// RPC calls are not allowed in Local mode.
IF stat.bLocal THEN
	RPC_MoveAbs	:= M_SetRpcStatus(E_MOTOR_RPC_ERROR.LOCAL);
	RETURN;
// Move Absolute command is accepted only in OP state.
ELSIF	stat.nState <> E_MOTOR_STATE.OP	THEN
	RPC_MoveAbs	:= M_SetRpcStatus(E_MOTOR_RPC_ERROR.NOT_OP);
	RETURN;
// Set velocity cannot be <=0.0.
ELSIF	in_lrVel <= 0.0	THEN
	RPC_MoveAbs	:= M_SetRpcStatus(E_MOTOR_RPC_ERROR.VEL_NEG);
	RETURN;
// Set velocity cannot be greater than MAX Velocity.
ELSIF	in_lrVel > stat.axis.lrMaxVelocity	THEN
	RPC_MoveAbs	:= M_SetRpcStatus(E_MOTOR_RPC_ERROR.VEL_MAX);
	RETURN;
// If SW limits are active, check the limits
ELSIF cfg.lrMinPosition <> 0.0 OR cfg.lrMaxPosition <> 0.0 THEN
	IF in_lrPos < cfg.lrMinPosition THEN
		RPC_MoveAbs	:= M_SetRpcStatus(E_MOTOR_RPC_ERROR.SW_LIMIT_LOWER);
		RETURN;
	ELSIF in_lrPos > cfg.lrMaxPosition THEN
		RPC_MoveAbs	:= M_SetRpcStatus(E_MOTOR_RPC_ERROR.SW_LIMIT_UPPER);
		RETURN;
	END_IF
END_IF

// Set command
ctrl.nCommand 		:= E_MOTOR_COMMAND.MOTOR_MOVE;
ctrl.nMoveType		:= E_MOTOR_MOVE_TYPE.ABSOLUTE;
ctrl.lrPosition		:= in_lrPos;
ctrl.lrVelocity		:= in_lrVel;
ctrl.bExecute 		:= TRUE;

// Call was successful
RPC_MoveAbs	:= M_SetRpcStatus(E_MOTOR_RPC_ERROR.OK);
END_METHOD

{attribute 'TcRpcEnable':='1'}
METHOD RPC_MoveRel : INT
VAR_INPUT
	in_lrPos:	LREAL;
	in_lrVel:	LREAL;
END_VAR
// If unsafe, move is not allowed.
IF NOT in_bSafe THEN
	RPC_MoveRel	:= M_SetRpcStatus(E_MOTOR_RPC_ERROR.UNSAFE);
	RETURN;
END_IF

// RPC calls are not allowed in Local mode.
IF stat.bLocal THEN
	RPC_MoveRel	:= M_SetRpcStatus(E_MOTOR_RPC_ERROR.LOCAL);
	RETURN;
// Move Relative command is accepted only in OP state.
ELSIF	stat.nState <> E_MOTOR_STATE.OP	THEN
	RPC_MoveRel	:= M_SetRpcStatus(E_MOTOR_RPC_ERROR.NOT_OP);
	RETURN;
// Set velocity cannot be <=0.0.
ELSIF	in_lrVel <= 0.0	THEN
	RPC_MoveRel	:= M_SetRpcStatus(E_MOTOR_RPC_ERROR.VEL_NEG);
	RETURN;
// Set velocity cannot be greater than MAX Velocity.
ELSIF	in_lrVel > stat.axis.lrMaxVelocity	THEN
	RPC_MoveRel	:= M_SetRpcStatus(E_MOTOR_RPC_ERROR.VEL_MAX);
	RETURN;
// If SW limits are active, check the limits
ELSIF cfg.lrMinPosition <> 0.0 OR cfg.lrMaxPosition <> 0.0 THEN
	IF (in_lrPos + stat.lrPosActual) < cfg.lrMinPosition THEN
		RPC_MoveRel	:= M_SetRpcStatus(E_MOTOR_RPC_ERROR.SW_LIMIT_LOWER);
		RETURN;
	ELSIF (in_lrPos + stat.lrPosActual) > cfg.lrMaxPosition THEN
		RPC_MoveRel	:= M_SetRpcStatus(E_MOTOR_RPC_ERROR.SW_LIMIT_UPPER);
		RETURN;
	END_IF
END_IF

// Set command
ctrl.nCommand 		:= E_MOTOR_COMMAND.MOTOR_MOVE;
ctrl.nMoveType		:= E_MOTOR_MOVE_TYPE.RELATIVE;
ctrl.lrOffset		:= in_lrPos;
ctrl.lrVelocity		:= in_lrVel;
ctrl.bExecute 		:= TRUE;

// Call was successful
RPC_MoveRel	:= M_SetRpcStatus(E_MOTOR_RPC_ERROR.OK);
END_METHOD

{attribute 'TcRpcEnable':='1'}
METHOD RPC_MoveVel : INT
VAR_INPUT
	in_lrVel:	LREAL;
END_VAR
// If unsafe, move is not allowed.
IF NOT in_bSafe THEN
	RPC_MoveVel	:= M_SetRpcStatus(E_MOTOR_RPC_ERROR.UNSAFE);
	RETURN;
END_IF

// RPC calls are not allowed in Local mode.
IF stat.bLocal THEN
	RPC_MoveVel	:= M_SetRpcStatus(E_MOTOR_RPC_ERROR.LOCAL);
	RETURN;
END_IF

// Move in Velocity command is accepted only in OP state.
IF	stat.nState <> E_MOTOR_STATE.OP	THEN
	RPC_MoveVel	:= M_SetRpcStatus(E_MOTOR_RPC_ERROR.NOT_OP);
	RETURN;
// Set velocity cannot be 0.0.
ELSIF	in_lrVel = 0.0	THEN
	RPC_MoveVel	:= M_SetRpcStatus(E_MOTOR_RPC_ERROR.VEL_ZERO);
	RETURN;
// Set velocity cannot be greater than MAX Velocity.
// Note that MoveVel() accepts negative velocity. That is
// why we use ABS().
ELSIF	ABS(in_lrVel) > stat.axis.lrMaxVelocity	THEN
	RPC_MoveVel	:= M_SetRpcStatus(E_MOTOR_RPC_ERROR.VEL_MAX);
	RETURN;
ELSE
	// Set command
	ctrl.nCommand 		:= E_MOTOR_COMMAND.MOTOR_MOVE;
	ctrl.nMoveType		:= E_MOTOR_MOVE_TYPE.VELOCITY;
	
	// Set the direction of movement based on the velocity sign.
	// Velocity is always passed as positive.
	IF in_lrVel < 0.0 THEN
		ctrl.lrVelocity		:= -in_lrVel;
		ctrl.nDirection		:= MC_Negative_Direction;
	ELSE
		ctrl.lrVelocity		:= in_lrVel;
		ctrl.nDirection		:= MC_Positive_Direction;
	END_IF

	ctrl.bExecute 		:= TRUE;
	
	// Call was successful
	RPC_MoveVel	:= M_SetRpcStatus(E_MOTOR_RPC_ERROR.OK);
END_IF
END_METHOD

{attribute 'TcRpcEnable':='1'}
METHOD RPC_Reset : INT
VAR_INPUT
END_VAR
// RPC calls are not allowed in Local mode.
IF stat.bLocal THEN
	RPC_Reset	:= M_SetRpcStatus(E_MOTOR_RPC_ERROR.LOCAL);
	RETURN;
END_IF

ctrl.nCommand := E_MOTOR_COMMAND.RESET;
ctrl.bExecute := TRUE;

// Call was successful
RPC_Reset	:= M_SetRpcStatus(E_MOTOR_RPC_ERROR.OK);
END_METHOD

{attribute 'TcRpcEnable':='1'}
METHOD RPC_SetDebug : INT
VAR_INPUT
	in_bDebug:	BOOL 	:= FALSE;		// If TRUE, show event logs of Debug type
END_VAR
// Enable/disable Debugging
cfg.bDebug	:= in_bDebug;

// Call was successful
RPC_SetDebug	:= M_SetRpcStatus(E_MOTOR_RPC_ERROR.OK);
END_METHOD

{attribute 'TcRpcEnable':='1'}
METHOD RPC_SetLog : INT
VAR_INPUT
	in_bLog:	BOOL 	:= FALSE;		// If TRUE, activate event logging
END_VAR
// Enable/disable Logging
cfg.bLog	:= in_bLog;

// Call was successful
RPC_SetLog	:= M_SetRpcStatus(E_MOTOR_RPC_ERROR.OK);
END_METHOD

{attribute 'TcRpcEnable':='1'}
METHOD RPC_Stop : INT
VAR_INPUT
END_VAR
// RPC calls are not allowed in Local mode.
IF stat.bLocal THEN
	RPC_Stop	:= M_SetRpcStatus(E_MOTOR_RPC_ERROR.LOCAL);
	RETURN;
END_IF

ctrl.nCommand := E_MOTOR_COMMAND.STOP;
ctrl.bExecute := TRUE;

// Call was successful
RPC_Stop	:= M_SetRpcStatus(E_MOTOR_RPC_ERROR.OK);
END_METHOD

METHOD UserPostInit : BOOL
VAR_OUTPUT
	nErrorId:	E_MOTOR_ERROR	:= E_MOTOR_ERROR.OK;
END_VAR
VAR
END_VAR
// TODOUSER:
// Dummy implementation.
// Configure cfg.bExecUserPostInit to TRUE.
// Implement PostInit logic.
// If error, set error description in this method using M_SetError(nErrorId, ...) - see below.

stat.sStatus	:= 'User Post-Init Method';

IF Dummy_UserExample() THEN
	UserPostInit	:= TRUE;
	stat.sStatus	:= 'OK';
	RETURN;
END_IF

// Check if the timer has expired. If yes, we have a problem *)
toutCmd();
IF toutCmd.Q = TRUE THEN
	toutCmd(IN := FALSE);
	nErrorId := E_MOTOR_ERROR.TIMEOUT_USER_POSTINIT;
	M_SetError(nErrorId, 'ERROR: Timeout during USER POST INIT');
	UserPostInit	:= TRUE;	// Exit (with error)
	RETURN;
END_IF


(* Check for motion errors *)
IF Axis.Status.Error THEN
	nErrorId	:= UDINT_TO_INT(Axis.Status.ErrorID);
	M_SetError(nErrorId, 'ERROR: Axis error during USER POST INIT');
	UserPostInit	:= TRUE;	// Exit (with error)
	RETURN;
END_IF

// Dummy implementation.
// Dummy error for testing.
//nErrorId := E_MOTOR_ERROR.TIMEOUT;
//M_SetError(nErrorId, 'ERROR: Dummy error during USER POST INIT');
//UserPostInit	:= TRUE;
RETURN;
END_METHOD

METHOD UserPostMove : BOOL
VAR_OUTPUT
	nErrorId:	E_MOTOR_ERROR	:= E_MOTOR_ERROR.OK;
END_VAR
VAR
END_VAR
// TODOUSER:
// Dummy implementation.
// Configure cfg.bExecUserPostMove to TRUE.
// Implement PostMove logic.
// If error, set error description in this method using M_SetError(nErrorId, ...) - see below.

stat.sStatus	:= 'User Post-Move Method';

IF Dummy_UserExample() THEN
	UserPostMove	:= TRUE;
	stat.sStatus	:= 'OK';
	RETURN;
END_IF

// Check if the timer has expired. If yes, we have a problem *)
toutCmd();
IF toutCmd.Q = TRUE THEN
	toutCmd(IN := FALSE);
	nErrorId := E_MOTOR_ERROR.TIMEOUT_USER_POSTMOVE;
	M_SetError(nErrorId, 'ERROR: Timeout during USER POST MOVE');
	UserPostMove	:= TRUE;	// Exit (with error)
	RETURN;
END_IF


(* Check for motion errors *)
IF Axis.Status.Error THEN
	nErrorId	:= UDINT_TO_INT(Axis.Status.ErrorID);
	M_SetError(nErrorId, 'ERROR: Axis error during USER POST MOVE');
	UserPostMove	:= TRUE;	// Exit (with error)
	RETURN;
END_IF

// Dummy implementation.
// Dummy error for testing.
//nErrorId := E_MOTOR_ERROR.TIMEOUT;
//M_SetError(nErrorId, 'ERROR: Dummy error during USER POST MOVE');
//UserPostMove	:= TRUE;
RETURN;
END_METHOD

METHOD UserPreInit : BOOL
VAR_OUTPUT
	nErrorId:	E_MOTOR_ERROR	:= E_MOTOR_ERROR.OK;
END_VAR
VAR
END_VAR
// TODOUSER:
// Dummy implementation.
// Configure cfg.bExecUserPreInit to TRUE.
// Implement PreInit logic.
// If error, set error description in this method using M_SetError(nErrorId, ...) - see below.

stat.sStatus	:= 'User Pre-Init Method';

IF Dummy_UserExample() THEN
	UserPreInit	:= TRUE;
	stat.sStatus	:= 'OK';
	RETURN;
END_IF

// Check if the timer has expired. If yes, we have a problem *)
toutCmd();
IF toutCmd.Q = TRUE THEN
	toutCmd(IN := FALSE);
	nErrorId := E_MOTOR_ERROR.TIMEOUT_USER_PREINIT;
	M_SetError(nErrorId, 'ERROR: Timeout during USER PRE INIT');
	UserPreInit	:= TRUE;	// Exit (with error)
	RETURN;
END_IF


(* Check for motion errors *)
IF Axis.Status.Error THEN
	nErrorId	:= UDINT_TO_INT(Axis.Status.ErrorID);
	M_SetError(nErrorId, 'ERROR: Axis error during USER PRE INIT');
	UserPreInit	:= TRUE;	// Exit (with error)
	RETURN;
END_IF

// Dummy implementation.
// Dummy error for testing.
//nErrorId := E_MOTOR_ERROR.TIMEOUT;
//M_SetError(nErrorId, 'ERROR: Dummy error during USER PRE INIT');
//UserPreInit	:= TRUE;
RETURN;
END_METHOD

METHOD UserPreMove : BOOL
VAR_OUTPUT
	nErrorId:	E_MOTOR_ERROR	:= E_MOTOR_ERROR.OK;
END_VAR
VAR
END_VAR
// TODOUSER:
// Dummy implementation.
// Configure cfg.bExecUserPreMove to TRUE.
// Implement PreMove logic.
// If error, set error description in this method using M_SetError(nErrorId, ...) - see below.

stat.sStatus	:= 'User Pre-Move Method';

IF Dummy_UserExample() THEN
	UserPreMove		:= TRUE;
	stat.sStatus	:= 'OK';
	RETURN;
END_IF

// Check if the timer has expired. If yes, we have a problem *)
toutCmd();
IF toutCmd.Q = TRUE THEN
	toutCmd(IN := FALSE);
	nErrorId := E_MOTOR_ERROR.TIMEOUT_USER_PREMOVE;
	M_SetError(nErrorId, 'ERROR: Timeout during USER PRE MOVE');
	UserPreMove	:= TRUE;	// Exit (with error)
	RETURN;
END_IF


(* Check for motion errors *)
IF Axis.Status.Error THEN
	nErrorId	:= UDINT_TO_INT(Axis.Status.ErrorID);
	M_SetError(nErrorId, 'ERROR: Axis error during USER PRE MOVE');
	UserPreMove	:= TRUE;	// Exit (with error)
	RETURN;
END_IF

// Dummy implementation.
// Dummy error for testing.
//nErrorId := E_MOTOR_ERROR.TIMEOUT;
//M_SetError(nErrorId, 'ERROR: Dummy error during USER PRE MOVE');
//UserPreMove	:= TRUE;
RETURN;
END_METHOD

END_FUNCTION_BLOCK

// ---- POUs/Motor/FB_MOTOR_BASE.TcPOU
FUNCTION_BLOCK FB_MOTOR_BASE
VAR_INPUT
	// EICSSW-1923
	{attribute 'OPC.UA.DA' := '0'}
	in_bSafe:		BOOL	:= TRUE;	// Flag if safe to move the motor
	{attribute 'OPC.UA.DA' := '0'}
	in_bDisableIfUnsafe:	BOOL := FALSE;	// If unsafe, motor is disabled
END_VAR
VAR_OUTPUT
END_VAR
VAR RETAIN
END_VAR
VAR
	{attribute 'OPC.UA.DA' := '1'}
	cfg:		T_MOTOR_CFG;		// Config parameters
	{attribute 'OPC.UA.DA' := '1'}
	ctrl:		T_MOTOR_CTRL;		// Control parameters
	{attribute 'OPC.UA.DA' := '1'}
	{attribute 'OPC.UA.DA.Access' := '1'}
	info:		T_MOTOR_INFO;		// Driver Info - ReadOnly
	{attribute 'OPC.UA.DA' := '1'}
	{attribute 'OPC.UA.DA.Access' := '1'}
	stat:		T_MOTOR_STAT;		// Status parameters - ReadOnly

	{attribute 'OPC.UA.DA' := '0'}
	nEvent:		      	DINT := E_MOTOR_EVENT.NONE;
	{attribute 'OPC.UA.DA' := '0'}
	nInternalEvent:		DINT := E_MOTOR_EVENT.NONE;
	
	// Operational Events
	{attribute 'OPC.UA.DA' := '0'}
	fbEventStart:	FB_TcMessage;
	{attribute 'OPC.UA.DA' := '0'}
	fbEventEnd:		FB_TcMessage;
	{attribute 'OPC.UA.DA' := '0'}
	fbEventError:	FB_TcMessage;
	{attribute 'OPC.UA.DA' := '0'}
	fbEventDebug:	FB_TcMessage;
	{attribute 'OPC.UA.DA' := '0'}
	fbEventGeneral:	FB_TcMessage;
	{attribute 'OPC.UA.DA' := '0'}
	fbEventMoveAbs:	FB_TcMessage;
	{attribute 'OPC.UA.DA' := '0'}
	fbEventMoveRel:	FB_TcMessage;
	{attribute 'OPC.UA.DA' := '0'}
	fbEventMoveVel:	FB_TcMessage;
	
	(***** Physical signals - to be mapped!!! *****)

	(* Outputs *)

	(* Inputs *)
	

END_VAR

METHOD ActionClearNOVRAM
VAR_INPUT
END_VAR
END_METHOD

METHOD ActionEnableExecute
VAR_INPUT
END_VAR
END_METHOD

METHOD ActionErrExecute
VAR
END_VAR
END_METHOD

METHOD ActionInitAbort
VAR_INPUT
END_VAR
END_METHOD

METHOD ActionInitComplete
VAR_INPUT
END_VAR
END_METHOD

METHOD ActionInitExecute
VAR_INPUT
END_VAR
END_METHOD

METHOD ActionInitReject
VAR_INPUT
END_VAR
END_METHOD

METHOD ActionMoveExecute
VAR_INPUT
END_VAR
END_METHOD

METHOD ActionResetExecute
VAR_INPUT
END_VAR
END_METHOD

METHOD ActionSetPosition
VAR_INPUT
END_VAR
END_METHOD

METHOD ActionStopExecute
VAR_INPUT
END_VAR
END_METHOD

METHOD ActionUnexpExecute
VAR_INPUT
END_VAR
END_METHOD

METHOD ActivityClearingNOVRAM
VAR_INPUT
END_VAR
END_METHOD

METHOD ActivityInitAborting
VAR_INPUT
END_VAR
END_METHOD

METHOD ActivityInitializing
VAR_INPUT
END_VAR
END_METHOD

METHOD ActivityMoving
VAR_INPUT
END_VAR
END_METHOD

METHOD ActivitySettingPosition
VAR_INPUT
END_VAR
END_METHOD

METHOD ActivityStopping
VAR_INPUT
END_VAR
END_METHOD

METHOD CheckForEvents
VAR_INPUT
END_VAR
END_METHOD

METHOD M_CheckDisableIfUnsafe
VAR_INPUT
END_VAR
IF NOT in_bSafe AND in_bDisableIfUnsafe	THEN
	IF stat.bEnabled	THEN
		stat.bEnabled	:= FALSE;
		M_LogEventGeneral('Not safe to move. Motor disabled.');
	END_IF
END_IF
END_METHOD

METHOD M_GetErrorText : STRING
VAR_INPUT
	nErrorID:	DINT;
END_VAR
VAR
	str:	STRING;
END_VAR
			
CASE nErrorID OF
	E_MOTOR_ERROR.OK:						str	:= 'OK';
	E_MOTOR_ERROR.HW_NOT_OP:				str	:= 'ERROR: TwinCAT not OP or CouplerState not mapped.';
	E_MOTOR_ERROR.LOCAL:					str	:= 'ERROR: Control not allowed. Motor in Local mode.';
	E_MOTOR_ERROR.INIT_ABORTED:				str	:= 'ERROR: INIT command aborted.';
	E_MOTOR_ERROR.TIMEOUT_INIT:				str	:= 'ERROR: INIT timed out.';
	E_MOTOR_ERROR.TIMEOUT_MOVE:				str	:= 'ERROR: Move timed out.';
	E_MOTOR_ERROR.TIMEOUT_RESET:			str	:= 'ERROR: Reset timed out.';
	E_MOTOR_ERROR.TIMEOUT_SETPOS:			str	:= 'ERROR: Set Position timed out.';
	E_MOTOR_ERROR.TIMEOUT_USER_PREINIT:		str	:= 'ERROR: User PRE-INIT timed out.';
	E_MOTOR_ERROR.TIMEOUT_USER_POSTINIT:	str	:= 'ERROR: User POST-INIT timed out.';
	E_MOTOR_ERROR.TIMEOUT_USER_PREMOVE:		str	:= 'ERROR: User PRE-MOVE timed out.';
	E_MOTOR_ERROR.TIMEOUT_USER_POSTMOVE:	str	:= 'ERROR: User POST-MOVE timed out.';
	E_MOTOR_ERROR.SETPOS:					str	:= 'ERROR: Set Position failed.';
	E_MOTOR_ERROR.STOP:						str	:= 'ERROR: STOP failed.';
	
	E_MOTOR_ERROR.ABORT:					str	:= 'ERROR: Motion aborted.';
	E_MOTOR_ERROR.SW_LIMIT_LOWER:			str	:= 'ERROR: Lower SW Limit Exceeded.';
	E_MOTOR_ERROR.SW_LIMIT_UPPER:			str	:= 'ERROR: Upper SW Limit Exceeded.';
	E_MOTOR_ERROR.BRAKE_ACTIVE:				str	:= 'ERROR: Cannot move. Brake active.';
	E_MOTOR_ERROR.BRAKE_ENGAGE:				str	:= 'ERROR: Failed to engage brake.';
	E_MOTOR_ERROR.BRAKE_DISENGAGE:			str	:= 'ERROR: Failed to disengage brake.';
	E_MOTOR_ERROR.SWITCH_NOT_USED:			str	:= 'ERROR: Switch was not detected in previous INIT action.';
	E_MOTOR_ERROR.ENABLE:					str	:= 'ERROR: Failed to enable Axis.';
	E_MOTOR_ERROR.NOVRAM_READ:				str	:= 'ERROR: Failed to read from NOVRAM';
	E_MOTOR_ERROR.NOVRAM_WRITE:				str	:= 'ERROR: Failed to write to NOVRAM';
	E_MOTOR_ERROR.SWITCH_EXIT:				str	:= 'ERROR: Timeout on switch exit. Check nTimeoutSwitch.';
	E_MOTOR_ERROR.STOP_LIMITS_BOTH:			str	:= 'ERROR: Both LSTOP and USTOP limits active.';
	E_MOTOR_ERROR.HW_LIMITS_BOTH:			str	:= 'ERROR: Both limit switches LHW and UHW active.';
	E_MOTOR_ERROR.IN_POS:					str	:= 'ERROR: In-Pos switch not active at the end of movement.';
	E_MOTOR_ERROR.LOCKED:					str	:= 'ERROR: Motor Locked! Cannot move.';
	E_MOTOR_ERROR.SoE_ADS_ERROR:			str	:= 'ERROR: SoE ADS Error.';
	E_MOTOR_ERROR.SoE_SERCOS_ERROR:			str	:= 'ERROR: SoE Sercos Error.';
	E_MOTOR_ERROR.UNSAFE:					str	:= 'ERROR: Not safe to move.';

	E_MOTOR_ERROR.SIM_NOT_INITIALISED:		str	:= 'ERROR: Simulator not initialised.';
	E_MOTOR_ERROR.SIM_NULL_POINTER:			str	:= 'ERROR: Simulator input parameter is a NULL pointer.';
	
	// Beckhoff TwinCAT most common errors
	E_MOTOR_ERROR.TC_VEL:					str	:= 'ERROR: Requested set velocity is not allowed.';
	E_MOTOR_ERROR.TC_NOT_READY_FOR_START:	str	:= 'ERROR: Drive not ready during axis start.';
	E_MOTOR_ERROR.TC_DISABLED_MOVE:			str	:= 'ERROR: Motor disabled while moving. Reset required!';
	E_MOTOR_ERROR.TC_BISECTION:				str	:= 'WARNING: Motion command could not be realized (BISECTION)';
	E_MOTOR_ERROR.TC_MODULO_POS:			str	:= 'ERROR: Target position >= full turn (modulo-period)';
	E_MOTOR_ERROR.TC_STOP_ACTIVE:			str	:= 'ERROR: Stop command still active. Axis locked. Reset required!';
	E_MOTOR_ERROR.TC_VEL_NEG:				str	:= 'ERROR: Set velocity not allowed (<=0)';
	E_MOTOR_ERROR.TC_TARGET_LSW:			str	:= 'ERROR: Target position beyond Lower Software Limit.';
	E_MOTOR_ERROR.TC_TARGET_USW:			str	:= 'ERROR: Target position beyond Upper Software Limit.';
	E_MOTOR_ERROR.TC_FOLLOWING_ERROR:		str	:= 'ERROR: Following error. Reset required!';
	E_MOTOR_ERROR.TC_NOT_READY:				str	:= 'ERROR: Drive not ready for operation.';
	E_MOTOR_ERROR.TC_IN_POS_6_SEC:			str	:= 'ERROR: In-position 6 sec timeout. Reset required!';
ELSE
	IF nErrorID > 10000 THEN
		str	:= concat('Unregistered error: ', DINT_TO_STRING(nErrorID));
		str	:= concat(str, ' Check TwinCAT error codes.');
	ELSE
		str	:= 'Unregistered internal error. Report it to ESO.';
	END_IF
END_CASE

M_GetErrorText	:= str;
END_METHOD

METHOD M_GetLogicalState : BOOL
(*
	This method returns the state of the variable based on its 
	activeLow configuration.
	Syntax:
		bState	:= GetLogicalState (<var value>,  <activeLow cfg>);
		
	Example 1:
		var = TRUE;
		activeLow = FALSE;
		bState	:= GetLogicalState (TRUE,  FALSE); = TRUE

	Example 2:
		var = TRUE;
		activeLow = TRUE;
		bState	:= GetLogicalState (TRUE,  TRUE); = FALSE
*)
VAR_INPUT
	state:		BOOL;
	activeLow:	BOOL;
END_VAR
IF activeLow THEN
	M_GetLogicalState := NOT state;
ELSE
	M_GetLogicalState := state;
END_IF
END_METHOD

METHOD M_GetTimeInSec : UDINT
(*
	This method returns absolute time in seconds.
*)
VAR_INPUT
END_VAR
VAR
	fbGetSystemTime:	GETSYSTEMTIME;
	timeLoDW:			DWORD;
	timeHiDW:			DWORD;
	nSecondsLo:			UDINT;
	nSecondsHi:			UDINT;

END_VAR
fbGetSystemTime (timeLoDW => timeLoDW, timeHiDW => timeHiDW); (* System time is given in 100ns *)
nSecondsLo	:= DWORD_TO_UDINT(timeLoDW) / 10000000; (* Convert to seconds *)
(* One unit from HI WORD represents 16#FFFFFFFF/10000000 = 429.4967296 seconds *)
nSecondsHi	:= LREAL_TO_UDINT(DWORD_TO_LREAL(timeHiDW) * 429.4967296);

M_GetTimeInSec	:= nSecondsHi + nSecondsLo;
END_METHOD

METHOD M_LogEventDebug : BOOL
VAR_INPUT
	sText:	STRING	:= '';
END_VAR
// Log Debug events only if both logging and debugging are enabled AND it is not a tracking command
IF cfg.bLog AND cfg.bDebug AND NOT (ctrl.nMoveType = E_MOTOR_MOVE_TYPE.TRACKING) THEN
	fbEventDebug.ipArguments.Clear().AddString(sText);
	fbEventDebug.Send(0);
END_IF
END_METHOD

METHOD M_LogEventEnd : BOOL
VAR_INPUT
	sText:	STRING	:= '';
END_VAR
// Log only if logging is enabled AND it is not a tracking command
IF  NOT cfg.bLog OR ctrl.nMoveType = E_MOTOR_MOVE_TYPE.TRACKING THEN
	RETURN;
END_IF

fbEventEnd.ipArguments.Clear().AddString(sText);
fbEventEnd.Send(0);
END_METHOD

METHOD M_LogEventError : BOOL
VAR_INPUT
	sText:	STRING	:= '';
END_VAR
// Log only if logging is enabled
IF  NOT cfg.bLog THEN
	RETURN;
END_IF

fbEventError.ipArguments.Clear().AddString(sText);
fbEventError.Send(0);
END_METHOD

METHOD M_LogEventGeneral : BOOL
VAR_INPUT
	sText:	STRING	:= '';
END_VAR
// Log only if logging is enabled AND it is not a tracking command
IF  NOT cfg.bLog OR ctrl.nMoveType = E_MOTOR_MOVE_TYPE.TRACKING THEN
	RETURN;
END_IF

fbEventGeneral.ipArguments.Clear().AddString(sText);
fbEventGeneral.Send(0);
END_METHOD

METHOD M_LogEventMoveAbs : BOOL
VAR_INPUT
	lrPos:	LREAL;
	lrVel:	LREAL;
END_VAR
// Log only if logging is enabled AND it is not a tracking command
IF  NOT cfg.bLog OR ctrl.nMoveType = E_MOTOR_MOVE_TYPE.TRACKING THEN
	RETURN;
END_IF

fbEventMoveAbs.ipArguments.Clear().AddLReal(lrPos).AddLReal(lrVel);
fbEventMoveAbs.Send(0);
END_METHOD

METHOD M_LogEventMoveRel : BOOL
VAR_INPUT
	lrPosRel:	LREAL;
	lrPosAct:	LREAL;
	lrVel:		LREAL;
END_VAR
// Log only if logging is enabled AND it is not a tracking command
IF  NOT cfg.bLog OR ctrl.nMoveType = E_MOTOR_MOVE_TYPE.TRACKING THEN
	RETURN;
END_IF

fbEventMoveRel.ipArguments.Clear().AddLReal(lrPosRel).AddLReal(lrPosAct).AddLReal(lrVel);
fbEventMoveRel.Send(0);
END_METHOD

METHOD M_LogEventMoveVel : BOOL
VAR_INPUT
	lrVel:	LREAL;
	dir:	DINT;
END_VAR
VAR
	lrVelTmp:	LREAL;
END_VAR
// Log only if logging is enabled AND it is not a tracking command
IF  NOT cfg.bLog OR ctrl.nMoveType = E_MOTOR_MOVE_TYPE.TRACKING THEN
	RETURN;
END_IF

IF dir = MC_Negative_Direction THEN
	lrVelTmp	:= -lrVel;
ELSE
	lrVelTmp	:= +lrVel;
END_IF
fbEventMoveVel.ipArguments.Clear().AddLReal(lrVelTmp);
fbEventMoveVel.Send(0);
END_METHOD

METHOD M_LogEventStart : BOOL
VAR_INPUT
	sText:	STRING	:= '';
END_VAR
// Log only if logging is enabled AND it is not a tracking command
IF  NOT cfg.bLog OR ctrl.nMoveType = E_MOTOR_MOVE_TYPE.TRACKING THEN
	RETURN;
END_IF

fbEventStart.ipArguments.Clear().AddString(sText);
fbEventStart.Send(0);
END_METHOD

// This method copies the description of the first error that caused the failure.
// For example, in case of a failure during move, the error description
// is written into stat.sFirstError and then the motor is commanded to stop.
// At the end of the stop, stat.sFirstError will be copied into stat.sErrorText so
// the user can see the real reason for the failure.
METHOD M_ReportFirstError
VAR_INPUT
END_VAR
IF stat.sFirstError <> '' THEN
	stat.sErrorText	:= stat.sFirstError;	// Copy stored error
	stat.sFirstError:= '';					// Clear stored error
END_IF
END_METHOD

METHOD M_SetStatus
VAR_INPUT
	nErrorCode:	E_MOTOR_ERROR;
END_VAR
stat.nErrorCode 	:= nErrorCode;
stat.sErrorText 	:= M_GetErrorText(nErrorCode);

IF nErrorCode <> E_MOTOR_ERROR.OK THEN
	stat.sStatus	:= 'ERROR';
	stat.nStatus	:= E_MOTOR_STATUS.ERROR;
ELSE
	stat.sStatus	:= 'OK';
	stat.nStatus	:= E_MOTOR_STATUS.OK;
END_IF
END_METHOD

METHOD M_SetStatusDescription
VAR_INPUT
	nAxisStatus:	E_MOTOR_STATUS;	(* Status number *)
	sStatus:		STRING;			(* Status text, e.g. IDLE, BUSY, etc. *)
END_VAR
stat.nErrorCode		:= E_MOTOR_ERROR.OK;
stat.nStatus		:= nAxisStatus;
stat.sErrorText		:= 'OK';
stat.sStatus		:= sStatus;
END_METHOD

METHOD ProcessEvents
VAR_INPUT
END_VAR

VAR
END_VAR

(* 
	Before processing the event, execute the Do-Activity tasks. 
	Note that, in case of orthogonal regions, more than one Do-Activity 
	could run in the same PLC cycle.
	Note: Most of these activities have timeouts since they take time.
*)

IF stat.nSubstate = E_MOTOR_SUBSTATE.NOTOP_INITIALIZING THEN
	ActivityInitializing();
END_IF

IF stat.nSubstate = E_MOTOR_SUBSTATE.NOTOP_ABORTING THEN
	ActivityInitAborting();
END_IF

IF stat.nSubstate = E_MOTOR_SUBSTATE.NOTOP_CLEARING_NOVRAM THEN
	ActivityClearingNOVRAM();
END_IF

IF	stat.nSubstate = E_MOTOR_SUBSTATE.OP_MOVING	AND
	nEvent <> E_MOTOR_EVENT.STOP					THEN
	ActivityMoving();
END_IF

IF stat.nSubstate = E_MOTOR_SUBSTATE.OP_STOPPING THEN
	ActivityStopping();
END_IF

IF stat.nSubstate = E_MOTOR_SUBSTATE.OP_SETTING_POS THEN
	ActivitySettingPosition();
END_IF


(* 
	Evaluate state machine transitions.
*)

CASE stat.nState OF

//***********************************
// NOTOP
//***********************************
E_MOTOR_STATE.NOTOP:

	(* Transitions from NOTOP substates *)
	CASE stat.nSubstate OF
	
	E_MOTOR_SUBSTATE.NOTOP_NOTREADY:		
		// Update error description if pending.
		M_ReportFirstError();		
		IF nEvent = E_MOTOR_EVENT.RESET THEN
			ActionResetExecute();
			RETURN;
		ELSIF nEvent = E_MOTOR_EVENT.INIT THEN
			ActionInitExecute();
			M_SetStatus(E_MOTOR_ERROR.OK);
			SetState(E_MOTOR_STATE.NOTOP, E_MOTOR_SUBSTATE.NOTOP_INITIALIZING);
			RETURN;
		ELSIF nEvent = E_MOTOR_EVENT.CLEAR_NOVRAM THEN
			ActionClearNOVRAM();
			M_SetStatus(E_MOTOR_ERROR.OK);
			SetState(E_MOTOR_STATE.NOTOP, E_MOTOR_SUBSTATE.NOTOP_CLEARING_NOVRAM);
			RETURN;
		END_IF
		
	E_MOTOR_SUBSTATE.NOTOP_INITIALIZING:			
		IF nEvent = E_MOTOR_EVENT.UNSAFE THEN
			// Set the first error that caused the failure
			M_SetStatus(E_MOTOR_ERROR.UNSAFE);
			stat.sFirstError	:= M_GetErrorText(E_MOTOR_ERROR.UNSAFE);
			M_LogEventError(stat.sFirstError);
			ActionInitAbort();
			SetState(E_MOTOR_STATE.NOTOP, E_MOTOR_SUBSTATE.NOTOP_ABORTING);
			RETURN;
		END_IF

		IF 	nEvent = E_MOTOR_EVENT.STOP  	OR  
			nEvent = E_MOTOR_EVENT.RESET 	 	THEN
			ActionInitAbort();
			SetState(E_MOTOR_STATE.NOTOP, E_MOTOR_SUBSTATE.NOTOP_ABORTING);
			RETURN;
		ELSIF nEvent = E_MOTOR_EVENT.ERRINIT THEN
			// Error description is set in ActivityInitializing().
			SetState(E_MOTOR_STATE.NOTOP, E_MOTOR_SUBSTATE.NOTOP_ERROR);
			RETURN;
		ELSIF nEvent = E_MOTOR_EVENT.ERRBRAKE OR 
			  nEvent = E_MOTOR_EVENT.ERRRESET 	THEN
			SetState(E_MOTOR_STATE.NOTOP, E_MOTOR_SUBSTATE.NOTOP_ERROR);
			RETURN;
		ELSIF nEvent = E_MOTOR_EVENT.INITDONE THEN
			ActionInitComplete();
			SetState(E_MOTOR_STATE.NOTOP, E_MOTOR_SUBSTATE.NOTOP_READY);
			RETURN;
		END_IF
		
	E_MOTOR_SUBSTATE.NOTOP_ABORTING:			
		IF	nEvent = E_MOTOR_EVENT.STOPDONE OR 
			nEvent = E_MOTOR_EVENT.ERRSTOP 		THEN
			SetState(E_MOTOR_STATE.NOTOP, E_MOTOR_SUBSTATE.NOTOP_NOTREADY);
			RETURN;
		ELSIF nEvent = E_MOTOR_EVENT.RESET THEN
			ActionInitAbort();
			M_SetStatus(E_MOTOR_ERROR.OK);
			SetState(E_MOTOR_STATE.NOTOP, E_MOTOR_SUBSTATE.NOTOP_NOTREADY);
			RETURN;
		END_IF
		
	E_MOTOR_SUBSTATE.NOTOP_READY:			
		// Check if the motor should be disabled due to non-safe operation
		M_CheckDisableIfUnsafe();
	
		IF nEvent = E_MOTOR_EVENT.RESET THEN
			ActionResetExecute();
			SetState(E_MOTOR_STATE.NOTOP, E_MOTOR_SUBSTATE.NOTOP_NOTREADY);
			RETURN;
		ELSIF nEvent = E_MOTOR_EVENT.ERRFAULT THEN
			SetState(E_MOTOR_STATE.NOTOP, E_MOTOR_SUBSTATE.NOTOP_NOTREADY);			
			RETURN;
		ELSIF nEvent = E_MOTOR_EVENT.ENABLE THEN
			M_LogEventGeneral('ENABLE Executed');
			M_SetStatus(E_MOTOR_ERROR.OK);
			SetState(E_MOTOR_STATE.OP, E_MOTOR_SUBSTATE.OP_STANDSTILL);
			RETURN;
		END_IF

	E_MOTOR_SUBSTATE.NOTOP_ERROR:			
		// Update error description if pending.
		M_ReportFirstError();		
		// Check if the motor should be disabled due to non-safe operation
		M_CheckDisableIfUnsafe();
	
		IF nEvent = E_MOTOR_EVENT.RESET THEN
			ActionResetExecute();
			SetState(E_MOTOR_STATE.NOTOP, E_MOTOR_SUBSTATE.NOTOP_NOTREADY);
			RETURN;
		ELSIF nEvent = E_MOTOR_EVENT.INIT THEN
			ActionInitExecute();
			M_SetStatus(E_MOTOR_ERROR.OK);
			SetState(E_MOTOR_STATE.NOTOP, E_MOTOR_SUBSTATE.NOTOP_INITIALIZING);
			RETURN;
		END_IF
		
	END_CASE

	(* Transitions from NOTOP state *)
	IF nEvent = E_MOTOR_EVENT.STOP THEN
		// Nothing to do. Motor is already standing
		RETURN;
	ELSIF nEvent = E_MOTOR_EVENT.ERRHW THEN
		stat.bEnabled		:= FALSE;	// Disable motor
		stat.bInitialised	:= FALSE;	// The motor has to be re-initialised
		SetState(E_MOTOR_STATE.NOTOP, E_MOTOR_SUBSTATE.NOTOP_ERROR);
		RETURN;
	ELSIF nEvent = E_MOTOR_EVENT.ERRLOCAL THEN
		M_SetStatus(E_MOTOR_ERROR.LOCAL);
		RETURN;
	END_IF
	
//***********************************
// OPERATIONAL
//***********************************
E_MOTOR_STATE.OP:

	(* Transitions from OP substates *)
	CASE stat.nSubstate OF
	E_MOTOR_SUBSTATE.OP_STANDSTILL:			
		// Update error description if pending.
		M_ReportFirstError();	
		// Check if the motor should be disabled due to non-safe operation
		M_CheckDisableIfUnsafe();
	
		IF nEvent = E_MOTOR_EVENT.MOTOR_MOVE THEN
			ActionMoveExecute();
			SetState(E_MOTOR_STATE.OP, E_MOTOR_SUBSTATE.OP_MOVING);
			RETURN;
		ELSIF nEvent = E_MOTOR_EVENT.SET_POSITION THEN
			ActionSetPosition();
			SetState(E_MOTOR_STATE.OP, E_MOTOR_SUBSTATE.OP_SETTING_POS);
			RETURN;		
		ELSIF nEvent = E_MOTOR_EVENT.DISABLE THEN
			M_LogEventGeneral('DISABLE Executed');
			SetState(E_MOTOR_STATE.NOTOP, E_MOTOR_SUBSTATE.NOTOP_READY);
			RETURN;		
		ELSIF nEvent = E_MOTOR_EVENT.ERRFAULT THEN
			ActionErrExecute();
			SetState(E_MOTOR_STATE.OP, E_MOTOR_SUBSTATE.OP_ERROR);
			RETURN;				
		END_IF

	E_MOTOR_SUBSTATE.OP_MOVING:			
		IF nEvent = E_MOTOR_EVENT.UNSAFE THEN
			// Set the first error that caused the failure
			M_SetStatus(E_MOTOR_ERROR.UNSAFE);
			stat.sFirstError	:= M_GetErrorText(E_MOTOR_ERROR.UNSAFE);
			M_LogEventError(stat.sFirstError);
			ActionStopExecute();
			SetState(E_MOTOR_STATE.OP, E_MOTOR_SUBSTATE.OP_STOPPING);
			RETURN;
		END_IF

		IF nEvent = E_MOTOR_EVENT.MOTOR_MOVE THEN
			ActionMoveExecute();
			RETURN;
		ELSIF nEvent = E_MOTOR_EVENT.STOP OR nEvent = E_MOTOR_EVENT.ERRHW THEN
			ActionStopExecute();
			SetState(E_MOTOR_STATE.OP, E_MOTOR_SUBSTATE.OP_STOPPING);
			RETURN;				
		ELSIF 	nEvent = E_MOTOR_EVENT.TIMEOUT_MOVE 		OR 
				nEvent = E_MOTOR_EVENT.ERRUSERPREMOVE 	OR
				nEvent = E_MOTOR_EVENT.ERRUSERPOSTMOVE 	OR
				nEvent = E_MOTOR_EVENT.ERRTARGETPAR	 	THEN
			// M_SetStatus() is already called in ActivityMoving() or User Pre/Post Move.
			// We just want to stop the motor after the failure.
			// TODO
			ActionStopExecute();
			SetState(E_MOTOR_STATE.OP, E_MOTOR_SUBSTATE.OP_STOPPING);
			RETURN;				
		ELSIF 	nEvent = E_MOTOR_EVENT.ERRBRAKE	OR 
				nEvent = E_MOTOR_EVENT.ERRENABLE	OR 
				nEvent = E_MOTOR_EVENT.ERRINPOS	OR
				nEvent = E_MOTOR_EVENT.ERRLOCKED 		THEN
			// M_SetStatus() is called in ActivityMoving since there are many possible failures.
			// Just go to failure.
			// TODO
			SetState(E_MOTOR_STATE.OP, E_MOTOR_SUBSTATE.OP_ERROR);
			RETURN;
		ELSIF nEvent = E_MOTOR_EVENT.SW_LIMIT_LOWER THEN
			SetState(E_MOTOR_STATE.OP, E_MOTOR_SUBSTATE.OP_STANDSTILL);
			RETURN;
		ELSIF nEvent = E_MOTOR_EVENT.SW_LIMIT_UPPER THEN
			SetState(E_MOTOR_STATE.OP, E_MOTOR_SUBSTATE.OP_STANDSTILL);
			RETURN;
		ELSIF nEvent = E_MOTOR_EVENT.ERRFAULT THEN
			ActionErrExecute();
			SetState(E_MOTOR_STATE.OP, E_MOTOR_SUBSTATE.OP_ERROR);
			RETURN;				
		ELSIF nEvent = E_MOTOR_EVENT.MOVEDONE THEN
			// Log event
			M_LogEventEnd('MOVE');
			SetState(E_MOTOR_STATE.OP, E_MOTOR_SUBSTATE.OP_STANDSTILL);
			RETURN;
		END_IF
		
	E_MOTOR_SUBSTATE.OP_SETTING_POS:			
		IF nEvent = E_MOTOR_EVENT.SETPOSDONE THEN
			SetState(E_MOTOR_STATE.OP, E_MOTOR_SUBSTATE.OP_STANDSTILL);
			RETURN;
		ELSIF nEvent = E_MOTOR_EVENT.TIMEOUT_SETPOS THEN
			SetState(E_MOTOR_STATE.OP, E_MOTOR_SUBSTATE.OP_STANDSTILL);
			RETURN;
		END_IF
		
	E_MOTOR_SUBSTATE.OP_STOPPING:			
		IF nEvent = E_MOTOR_EVENT.STOPDONE THEN
			SetState(E_MOTOR_STATE.OP, E_MOTOR_SUBSTATE.OP_STANDSTILL);
			RETURN;
		ELSIF nEvent = E_MOTOR_EVENT.ERRFAULT THEN
			SetState(E_MOTOR_STATE.OP, E_MOTOR_SUBSTATE.OP_ERROR);
			RETURN;
		ELSIF nEvent = E_MOTOR_EVENT.ERRSTOP THEN
			SetState(E_MOTOR_STATE.OP, E_MOTOR_SUBSTATE.OP_ERROR);
			RETURN;
		END_IF
		
	E_MOTOR_SUBSTATE.OP_ERROR:	
		// Update error description if pending.
		M_ReportFirstError();		
		// Check if the motor should be disabled due to non-safe operation
		M_CheckDisableIfUnsafe();

		IF nEvent = E_MOTOR_EVENT.MOTOR_MOVE THEN
			ActionMoveExecute();
			SetState(E_MOTOR_STATE.OP, E_MOTOR_SUBSTATE.OP_MOVING);
			RETURN;			
		ELSIF nEvent = E_MOTOR_EVENT.DISABLE THEN
			M_LogEventGeneral('DISABLE Executed');
			SetState(E_MOTOR_STATE.NOTOP, E_MOTOR_SUBSTATE.NOTOP_READY);
			RETURN;		
		END_IF

	END_CASE
	
	(* Transitions from OP state *)
	IF nEvent = E_MOTOR_EVENT.ERRHW THEN
		stat.bEnabled		:= FALSE;	// Disable motor
		stat.bInitialised	:= FALSE;	// The motor has to be re-initialised
		SetState(E_MOTOR_STATE.NOTOP, E_MOTOR_SUBSTATE.NOTOP_ERROR);
		RETURN;
	ELSIF nEvent = E_MOTOR_EVENT.RESET THEN
		// TODO: Maybe accept only if not moving
		ActionResetExecute();
		SetState(E_MOTOR_STATE.NOTOP, E_MOTOR_SUBSTATE.NOTOP_NOTREADY);
		RETURN;
	ELSIF nEvent = E_MOTOR_EVENT.ERRLOCAL THEN
		M_SetStatus(E_MOTOR_ERROR.LOCAL);
		RETURN;
	END_IF
	
END_CASE

(* 
	"Global" internal transitions valid in any state should go here.
	They do not change the active state configuration. 
	They are evaluated after all the others transitions have been 
	considered.
*) 
IF nEvent = E_MOTOR_EVENT.RESET THEN
	ActionResetExecute();
	SetState(E_MOTOR_STATE.NOTOP, E_MOTOR_SUBSTATE.NOTOP_NOTREADY);
	RETURN;
ELSIF nEvent = E_MOTOR_EVENT.STOP THEN
	ActionStopExecute();
	SetState(E_MOTOR_STATE.OP, E_MOTOR_SUBSTATE.OP_STOPPING);
	RETURN;
END_IF
END_METHOD

METHOD SetAction
VAR_INPUT
	actionName:		STRING;
END_VAR


stat.sActionDesc := actionName;
END_METHOD

METHOD SetEvent
VAR_INPUT
	nEventId:			DINT;
END_VAR

nEvent := nEventId;

CASE nEventId OF
	E_MOTOR_EVENT.NONE:
		stat.sEventDesc := '';
		RETURN;
		
	E_MOTOR_EVENT.RESET:
		stat.sEventDesc := 'CMD RESET';
		RETURN;
	
	E_MOTOR_EVENT.INIT:
		stat.sEventDesc := 'CMD INIT';
		RETURN;

	E_MOTOR_EVENT.STOP:
		stat.sEventDesc := 'CMD STOP';
		RETURN;

	E_MOTOR_EVENT.ENABLE:
		stat.sEventDesc := 'CMD ENABLE';
		RETURN;

	E_MOTOR_EVENT.DISABLE:
		stat.sEventDesc := 'CMD DISABLE';
		RETURN;

	E_MOTOR_EVENT.MOTOR_MOVE:
		stat.sEventDesc := 'CMD MOVE';
		RETURN;

	E_MOTOR_EVENT.SET_POSITION:
		stat.sEventDesc := 'CMD SET POSITION';
		RETURN;

	E_MOTOR_EVENT.CLEAR_NOVRAM:
		stat.sEventDesc := 'CMD CLEAR NOVRAM';
		RETURN;

	E_MOTOR_EVENT.MOVEDONE:
		stat.sEventDesc := 'INT MOVEDONE';
		RETURN;
	
	E_MOTOR_EVENT.STOPDONE:
		stat.sEventDesc := 'INT STOPDONE';
		RETURN;
	
	E_MOTOR_EVENT.ENABLEDONE:
		stat.sEventDesc := 'INT ENABLEDONE';
		RETURN;
	
	E_MOTOR_EVENT.DISABLEDONE:
		stat.sEventDesc := 'INT DISABLEDONE';
		RETURN;
	
	E_MOTOR_EVENT.INITDONE:
		stat.sEventDesc := 'INT INITDONE';
		RETURN;
	
	E_MOTOR_EVENT.SETPOSDONE:
		stat.sEventDesc := 'INT SETPOSDONE';
		RETURN;
	
	E_MOTOR_EVENT.UNSAFE:
		stat.sEventDesc := 'EXT UNSAFE';
		RETURN;
	
	E_MOTOR_EVENT.HWOK:
		stat.sEventDesc := 'SIG HWOK';
		RETURN;

	E_MOTOR_EVENT.ERRHW:
		stat.sEventDesc := 'INT ERRHW';
		RETURN;

	E_MOTOR_EVENT.ERRLOCAL:
		stat.sEventDesc := 'INT ERRLOCAL';
		RETURN;

	E_MOTOR_EVENT.ERRFAULT:	
		stat.sEventDesc := 'INT ERRFAULT';
		RETURN;

	E_MOTOR_EVENT.ERRINIT:
		stat.sEventDesc := 'INT ERRINIT';
		RETURN;

	E_MOTOR_EVENT.ERRENABLE:
		stat.sEventDesc := 'INT ERRENABLE';
		RETURN;
	
	E_MOTOR_EVENT.ERRDISABLE:
		stat.sEventDesc := 'INT ERRDISABLE';
		RETURN;
	
	E_MOTOR_EVENT.ERRBRAKE:
		stat.sEventDesc := 'INT ERRBRAKE';
		RETURN;
	
	E_MOTOR_EVENT.ERRINPOS:
		stat.sEventDesc := 'INT ERRINPOS';
		RETURN;
	
	E_MOTOR_EVENT.ERRTARGETPAR:
		stat.sEventDesc := 'INT ERRTARGETPAR';
		RETURN;
	
END_CASE 

(* INTERNAL ERROR *)
stat.sEventDesc := 'UNKNOWN EVENT';
END_METHOD

METHOD SetState : BOOL
VAR_INPUT
	nState:			E_MOTOR_STATE;
	nSubstate:		E_MOTOR_SUBSTATE;
END_VAR
(* 
	Update State Machine active state configuration.
*)

IF nState <> E_MOTOR_STATE.NONE THEN
	stat.nState	:= nState;
END_IF
IF nSubstate <> E_MOTOR_SUBSTATE.NONE THEN
	stat.nSubstate	:= nSubstate;
END_IF

(* Update active state configuration description *)

IF nState = E_MOTOR_STATE.NOTOP THEN
	stat.sState	:= 'NOT OP';
ELSIF nState = E_MOTOR_STATE.OP THEN
	stat.sState	:= 'OPERATIONAL';
END_IF

IF nSubstate = E_MOTOR_SUBSTATE.NOTOP_NOTREADY THEN
	stat.sSubstate	:= 'NOT READY';
ELSIF nSubstate = E_MOTOR_SUBSTATE.NOTOP_INITIALIZING THEN
	stat.sSubstate	:= 'INITIALIZING';
ELSIF nSubstate = E_MOTOR_SUBSTATE.NOTOP_READY THEN
	stat.sSubstate	:= 'READY';
ELSIF nSubstate = E_MOTOR_SUBSTATE.NOTOP_ERROR THEN
	stat.sSubstate	:= 'ERROR';
ELSIF nSubstate = E_MOTOR_SUBSTATE.OP_STANDSTILL THEN
	stat.sSubstate	:= 'STANDSTILL';
ELSIF nSubstate = E_MOTOR_SUBSTATE.OP_SETTING_POS THEN
	stat.sSubstate	:= 'SETTING POS';
ELSIF nSubstate = E_MOTOR_SUBSTATE.OP_MOVING THEN
	stat.sSubstate	:= 'MOVING';
ELSIF nSubstate = E_MOTOR_SUBSTATE.OP_STOPPING THEN
	stat.sSubstate	:= 'STOPPING';
ELSIF nSubstate = E_MOTOR_SUBSTATE.OP_ERROR THEN
	stat.sSubstate	:= 'ERROR';
ELSE
	stat.sSubstate	:= '';
END_IF


SetState	:= TRUE;
END_METHOD

METHOD SetStatus
VAR_INPUT
	nErrorCode:	E_MOTOR_ERROR;
	sErrorText:	STRING;
END_VAR
stat.nErrorCode 	:= nErrorCode;
stat.sErrorText 	:= sErrorText;

IF nErrorCode <> E_MOTOR_ERROR.OK THEN
	stat.sStatus	:= 'ERROR';
	stat.nStatus	:= E_MOTOR_STATUS.ERROR;
ELSE
	stat.sStatus	:= 'OK';
	stat.nStatus	:= E_MOTOR_STATUS.OK;
END_IF
END_METHOD

END_FUNCTION_BLOCK

// ---- POUs/Motor/FB_SIM_MOTOR.TcPOU
FUNCTION_BLOCK FB_SIM_MOTOR
VAR_INPUT
	ptrCfg:		POINTER TO T_MOTOR_CFG;
	ptrStat:	POINTER TO T_MOTOR_STAT;
END_VAR
VAR_OUTPUT
END_VAR
VAR
	{attribute 'OPC.UA.DA':='1'}
	cfg:			T_SIM_MOTOR_CFG;	(* ActiveLow configuration for each signal *)
	{attribute 'OPC.UA.DA':='1'}
	stat:			T_SIM_MOTOR_STAT;	(* Simulator status parameters *)
	
	{attribute 'OPC.UA.DA':='0'}
//	nCouplerState:	UINT := 8;       // normal coupler state
	
    (* Inputs *)
	{attribute 'OPC.UA.DA':='0'}
	i_bBrake_Ctrl	AT %I*:	BOOL;				(* Brake control signal - to be linked to q_bBrake_Ctrl *)

	(* Outputs *)	
	{attribute 'OPC.UA.DA':='0'}
	switches		AT %Q*:	T_MOTOR_SWITCHES;	(* Limit switches - to be linked to real Motor switches *)
	{attribute 'OPC.UA.DA':='0'}
	q_bBrake_Stat	AT %Q*:	BOOL;				(* Brake feedback signal - to be linked to i_bBrake_Stat  *)
	{attribute 'OPC.UA.DA':='0'}
	q_nCouplerState AT %Q*:		UINT := 8;		(* HW state - to be linked to i_nCouplerState *)
	
	{attribute 'OPC.UA.DA':='0'}
	timer_SwitchOn:		TON;
	{attribute 'OPC.UA.DA':='0'}
	timer_SwitchOff:	TON;
	{attribute 'OPC.UA.DA':='0'}
	timer_Brake:	TON;
	{attribute 'OPC.UA.DA':='0'}
	trgBrake:		R_TRIG;	// Trigger for brake activation
	{attribute 'OPC.UA.DA':='0'}
	trgInitCmd:		R_TRIG;	// Trigger for INIT command
	{attribute 'OPC.UA.DA':='0'}
	trgInitAction:	R_TRIG;	// Trigger for INIT action, e.g. FIND LHW
	
	// Action delays
//	nDelay_SwitchFind:		UDINT := 5000;	// 5 sec delay for finding switch
//	nDelay_SwitchActive:	UDINT := 7000;	// 7 sec delay for switch being active (exiting switch)
//	nDelay_Brake:			UDINT :=  500;	// 0.5 sec delay for brake activation
	
	{attribute 'OPC.UA.DA':='0'}
	nInitAction:	DINT := 0;		// No action yet
	{attribute 'OPC.UA.DA':='0'}
	bBrake:			BOOL := FALSE;
	
END_VAR

// Check for NULL pointers in input parameters.
// We cannot continue if any of the pointers is NULL.
IF ptrCfg = 0  OR  ptrStat = 0 THEN
	stat.nErrorCode	:= E_MOTOR_ERROR.SIM_NULL_POINTER;
	stat.sErrorText	:= 'ERROR: Input parameter is a NULL pointer';
	stat.sStatus	:= 'ERROR';
	RETURN;
END_IF

//
// When the simulator starts, all switches are clear and brakes are disengaged.
//
IF NOT stat.bInitialised THEN
	// Copy the real motor configuration
	RPC_ResetConfig();
	
	// Release brakes
	// The control signal for brakes MUST be active low - it's hard-coded in FB_MOTOR.
	// Therefore the feedback should use the inverse of i_bBrake_Ctrl.
	// Feedback active low is configured with bActiveLowBrake.
	// q_bBrake_Stat is the simulated feedback to the real motor.
	bBrake 			:= i_bBrake_Ctrl;
	q_bBrake_Stat	:= GetLogicalState(NOT i_bBrake_Ctrl, ptrCfg^.bActiveLowBrake);
	
	stat.nErrorCode		:= E_MOTOR_ERROR.OK;
	stat.sErrorText		:= 'OK';
	stat.sStatus		:= 'OK';
	stat.bInitialised	:= TRUE;
END_IF

// If the motor is not initialised and not enabled, reset simulator configuration.
// This way we avoid deadlock in case both limit switches (HW or STOP) are active.
IF 	NOT ptrStat^.bInitialised	AND 
	NOT ptrStat^.bEnabled 		AND
	((ptrStat^.signals[0].bActive AND ptrStat^.signals[5].bActive) OR
	 (ptrStat^.signals[1].bActive AND ptrStat^.signals[4].bActive)) THEN
	// Copy the real motor configuration
	RPC_ResetConfig();
END_IF


//
// Wait for events
// They can be:
// - New INIT sequence action that envolves activation of limit switches, e.g. FIND LHW.
// - Brake control change, i.e. apply or release.
//

//////////////////////////////
// Handling of limit switches
//////////////////////////////

// Checking for INIT command.
// The substate string will become 'INITIALIZING'.
// At this point, new configuration is written to the PLC.
// Copy it to the simulator.
trgInitCmd(CLK:=(ptrStat^.sSubstate = 'INITIALIZING'));
IF trgInitCmd.Q THEN
	// Copy the real motor configuration
	RPC_ResetConfig();
END_IF

// Clear REF switch at the end of INIT since it remains active in the FIND_REF_LE case.
IF ptrStat^.bInitialised AND ptrStat^.sStatus = 'STANDING' THEN
	switches.bREF	:= GetLogicalState(FALSE, cfg.bArrActiveLow[2].bValue);
END_IF

// Checking for INIT actions that require activation of limit switches
trgInitAction(CLK:=(nInitAction <> ptrStat^.nInitAction));
IF trgInitAction.Q THEN
	// Assign the current value, so we could detect next change.
	nInitAction := ptrStat^.nInitAction;	
	IF	nInitAction = MOTOR_INIT_ACTION_FIND_INDEX 	OR
		nInitAction = MOTOR_INIT_ACTION_FIND_REF_LE OR
		nInitAction = MOTOR_INIT_ACTION_FIND_REF_UE OR
		nInitAction = MOTOR_INIT_ACTION_FIND_LHW 	OR
		nInitAction = MOTOR_INIT_ACTION_FIND_UHW 	THEN 
		// Delay activation of the corresponding switch by nDelay_SwitchFind ms.
		timer_SwitchOn(IN:=FALSE);
		timer_SwitchOn(IN:=TRUE,PT:=UDINT_TO_TIME(cfg.nDelay_SwitchFind));
		
		IF nInitAction = MOTOR_INIT_ACTION_FIND_REF_LE THEN
			switches.bREF	:= GetLogicalState(TRUE, cfg.bArrActiveLow[2].bValue);
		END_IF
	END_IF
END_IF


// Switch activation
timer_SwitchOn();
IF timer_SwitchOn.Q THEN
	// Reset the timer.
	timer_SwitchOn(IN:=FALSE);
	CASE nInitAction OF
		// Activate the corresponding switch based on the INIT action.
		MOTOR_INIT_ACTION_FIND_INDEX:
			switches.bINDEX	:= GetLogicalState(TRUE, cfg.bArrActiveLow[3].bValue);
		MOTOR_INIT_ACTION_FIND_REF_LE:
			switches.bREF	:= GetLogicalState(FALSE, cfg.bArrActiveLow[2].bValue);
		MOTOR_INIT_ACTION_FIND_REF_UE:
			switches.bREF	:= GetLogicalState(TRUE, cfg.bArrActiveLow[2].bValue);
		MOTOR_INIT_ACTION_FIND_LHW:
			switches.bLHW	:= GetLogicalState(TRUE, cfg.bArrActiveLow[1].bValue);
		MOTOR_INIT_ACTION_FIND_UHW:
			switches.bUHW	:= GetLogicalState(TRUE, cfg.bArrActiveLow[4].bValue);
	END_CASE

	// Delay deactivation of the corresponding switch by nDelay_SwitchActive ms,
	// i.e. keep the switch active for nDelay_SwitchActive ms.
	timer_SwitchOff(IN:=FALSE);
	timer_SwitchOff(IN:=TRUE,PT:=UDINT_TO_TIME(cfg.nDelay_SwitchActive));
END_IF

// Switch deactivation
timer_SwitchOff();
IF timer_SwitchOff.Q THEN
	timer_SwitchOff(IN:=FALSE);
	// Deactivate the switch based on the INIT action.
	CASE nInitAction OF
		MOTOR_INIT_ACTION_FIND_INDEX:
			switches.bINDEX	:= GetLogicalState(FALSE, cfg.bArrActiveLow[3].bValue);
		MOTOR_INIT_ACTION_FIND_REF_LE:
			switches.bREF	:= GetLogicalState(TRUE, cfg.bArrActiveLow[2].bValue);
		MOTOR_INIT_ACTION_FIND_REF_UE:
			switches.bREF	:= GetLogicalState(FALSE, cfg.bArrActiveLow[2].bValue);
		MOTOR_INIT_ACTION_FIND_LHW:
			switches.bLHW	:= GetLogicalState(FALSE, cfg.bArrActiveLow[1].bValue);
		MOTOR_INIT_ACTION_FIND_UHW:
			switches.bUHW	:= GetLogicalState(FALSE, cfg.bArrActiveLow[4].bValue);
	END_CASE
END_IF


//////////////////////////////
// Handling of brakes
//////////////////////////////

IF ptrCfg^.bUseBrake THEN
	// Checking for the change in brake control signal
	trgBrake(CLK:=(bBrake <> i_bBrake_Ctrl));
	IF trgBrake.Q THEN
		// Assign the current value, so we could detect next change.
		bBrake := i_bBrake_Ctrl;
		// Bring the brake to set state after the delay of nDelay_Brake ms.
		timer_Brake(IN:=FALSE);
		timer_Brake(IN:=TRUE,PT:=UDINT_TO_TIME(cfg.nDelay_Brake));
	END_IF
	
	timer_Brake();
	IF timer_Brake.Q THEN
		// Reset timer for brake actions
		timer_Brake(IN:=FALSE);
		// The control signal for brakes MUST be active low.
		// Therefore the feedback should use the inverse of i_bBrake_Ctrl.
		// Feedback active low is configured with bActiveLowBrake.
		q_bBrake_Stat	:= GetLogicalState(NOT i_bBrake_Ctrl, cfg.bActiveLowBrake);
	END_IF
ELSE
	ptrCfg^.bActiveLowBrake	:= FALSE;
	cfg.bActiveLowBrake		:= FALSE;
	q_bBrake_Stat			:= GetLogicalState(FALSE, cfg.bActiveLowBrake);
END_IF

q_nCouplerState	:= cfg.nCouplerState;	// Set coupler state output

METHOD GetLogicalState : BOOL
(*
	This method returns the state of the variable based on its 
	activeLow configuration.
	Syntax:
		bState	:= GetLogicalState (<var value>,  <activeLow cfg>);
		
	Example 1:
		var = TRUE;
		activeLow = FALSE;
		bState	:= GetLogicalState (TRUE,  FALSE); = TRUE

	Example 2:
		var = TRUE;
		activeLow = TRUE;
		bState	:= GetLogicalState (TRUE,  TRUE); = FALSE
*)
VAR_INPUT
	state:		BOOL;
	activeLow:	BOOL;
END_VAR
IF activeLow THEN
	GetLogicalState := NOT state;
ELSE
	GetLogicalState := state;
END_IF
END_METHOD

{attribute 'TcRpcEnable':='1'}
METHOD RPC_ResetConfig : INT
VAR_INPUT
END_VAR
// Copy relevant configuration to the simulator
cfg.bArrActiveLow	:= ptrCfg^.bArrActiveLow;
cfg.bUseBrake		:= ptrCfg^.bUseBrake;
cfg.bActiveLowBrake	:= ptrCfg^.bActiveLowBrake;

// Deactivate simulated limit switches
switches.bLSTOP	:= GetLogicalState(FALSE, cfg.bArrActiveLow[0].bValue);
switches.bLHW	:= GetLogicalState(FALSE, cfg.bArrActiveLow[1].bValue);
switches.bREF	:= GetLogicalState(FALSE, cfg.bArrActiveLow[2].bValue);
switches.bINDEX	:= GetLogicalState(FALSE, cfg.bArrActiveLow[3].bValue);
switches.bUHW	:= GetLogicalState(FALSE, cfg.bArrActiveLow[4].bValue);
switches.bUSTOP	:= GetLogicalState(FALSE, cfg.bArrActiveLow[5].bValue);

	
IF NOT cfg.bUseBrake THEN
	// Brakes not used.
	// Setting bActiveLowBrake to TRUE would just confuse the user.
	// Clear the flag.
	ptrCfg^.bActiveLowBrake	:= FALSE;
	cfg.bActiveLowBrake		:= FALSE;
	// Brakes released
	q_bBrake_Stat	:= GetLogicalState(FALSE, ptrCfg^.bActiveLowBrake);
ELSE
	// Remember current brake state.
	// Use to detect change in brake control signal.
	bBrake			:= i_bBrake_Ctrl;
	// Brakes released
	q_bBrake_Stat	:= GetLogicalState(FALSE, ptrCfg^.bActiveLowBrake);
END_IF

// Reset INIT action recognition
trgInitAction(CLK:=FALSE);

cfg.nCouplerState	:= 8;
nInitAction			:= 0;

RPC_ResetConfig	:= E_MOTOR_RPC_ERROR.OK;
END_METHOD

{attribute 'TcRpcEnable':='1'}
METHOD RPC_SetCouplerState : INT
VAR_INPUT
	nValue:	UINT;	// Coupler state. 8=OP, any other value is a ERROR, i.e. NON_OP
END_VAR
cfg.nCouplerState	:= nValue;

RPC_SetCouplerState	:= E_MOTOR_RPC_ERROR.OK;
END_METHOD

{attribute 'TcRpcEnable':='1'}
METHOD RPC_SetDelay_Brake : INT
VAR_INPUT
	nDelay:	UDINT;
END_VAR
cfg.nDelay_Brake	:= nDelay;

RPC_SetDelay_Brake	:= E_MOTOR_RPC_ERROR.OK;
END_METHOD

{attribute 'TcRpcEnable':='1'}
METHOD RPC_SetDelay_SwitchActive : INT
VAR_INPUT
	nDelay:	UDINT;
END_VAR
cfg.nDelay_SwitchActive	:= nDelay;

RPC_SetDelay_SwitchActive:= E_MOTOR_RPC_ERROR.OK;
END_METHOD

{attribute 'TcRpcEnable':='1'}
METHOD RPC_SetDelay_SwitchFind : INT
VAR_INPUT
	nDelay:	UDINT;
END_VAR
cfg.nDelay_SwitchFind	:= nDelay;

RPC_SetDelay_SwitchFind	:= E_MOTOR_RPC_ERROR.OK;
END_METHOD

{attribute 'TcRpcEnable':='1'}
METHOD RPC_SetFailure_BrakeFeedback : INT
VAR_INPUT
END_VAR
// Execute only if brakes are used
IF cfg.bUseBrake THEN
	// Swap brake active low level in order to cause failure
	cfg.bActiveLowBrake	:= NOT ptrCfg^.bActiveLowBrake;
END_IF

RPC_SetFailure_BrakeFeedback	:= E_MOTOR_RPC_ERROR.OK;
END_METHOD

END_FUNCTION_BLOCK

// ---- POUs/MultiAxis/FB_MA_ADC.TcPOU
FUNCTION_BLOCK FB_MA_ADC EXTENDS FB_MA_BASE
VAR_INPUT
	{attribute 'OPC.UA.DA' := '0'}
	sMotorAdc1:			STRING	:= 'MotorAdc1';	(* Default Motor name *)
	{attribute 'OPC.UA.DA' := '0'}
	sMotorAdc2:			STRING	:= 'MotorAdc2';	(* Default Motor name *)
	
	{attribute 'OPC.UA.DA' := '0'}
	stSiteConstants:      T_ASTRO_SITE_CONSTANTS;
	
	{attribute 'OPC.UA.DA' := '0'}
	stEnvironmentData:    T_ASTRO_ENVIRONMENT;  
	
	{attribute 'OPC.UA.DA' := '0'}
	stPointingKernel:    T_ASTRO_POINTING_KERNEL_POSITIONS;  
	
	{attribute 'OPC.UA.DA' := '0'}
	nNOVRAM_DevId:	UDINT	:= 0;		(* NOVRAM device ID - normally 4 *)
	{attribute 'OPC.UA.DA' := '0'}
	nNOVRAM_Offset1:	UDINT	:= 0;		(* NOVRAM offset where ADC motor1 configuration is stored *)
	{attribute 'OPC.UA.DA' := '0'}
	nNOVRAM_Offset2:	UDINT	:= 0;		(* NOVRAM offset where ADC motor2 configuration is stored *)
	
END_VAR
VAR_OUTPUT
END_VAR
VAR
	
	{attribute 'OPC.UA.DA' := '1'}
	cfg:				T_ADC_CFG;
	{attribute 'OPC.UA.DA' := '1'}
	ctrl:				T_ADC_CTRL;
	{attribute 'OPC.UA.DA' := '1'}
	stat:				T_ADC_STAT;
	
	{attribute 'OPC.UA.DA':='1'}
	motor1:              FB_MOTOR;
	{attribute 'OPC.UA.DA':='1'}
	motor2:              FB_MOTOR;
	
	
END_VAR

// A MUST !!! Set references to real structures
RefCfg		REF=cfg;
RefCtrl		REF=ctrl;
RefStat		REF=stat;

motor1(	sName 				:= sMotorAdc1,
		in_bSafe			:= in_bSafe,
		in_bDisableIfUnsafe	:= in_bDisableIfUnsafe,
		nNOVRAM_DevId		:= nNOVRAM_DevId, 
		nNOVRAM_Offset		:= nNOVRAM_Offset1);
		
motor2(	sName 				:= sMotorAdc2,	
		in_bSafe			:= in_bSafe,
		in_bDisableIfUnsafe	:= in_bDisableIfUnsafe,
		nNOVRAM_DevId		:= nNOVRAM_DevId, 
		nNOVRAM_Offset		:= nNOVRAM_Offset2);

SUPER^(nNumAxes:=2, pMotor1:=ADR(motor1), pMotor2:=ADR(motor2));

METHOD M_LogCommand : BOOL
VAR
	cmd:	INT;
	mode:	int;
END_VAR
cmd		:= RefCtrl.nCommand;
mode	:= ctrl.nMode;

// Log ADC command.
// Set motor logging to FALSE when tracking,
// in order to reduce flooding of logs.
IF cmd = E_MA_COMMAND.RESET THEN
	pMotor1^.RPC_SetLog(TRUE);
	pMotor2^.RPC_SetLog(TRUE);
	M_SetStatus('Resetting ADC device...');		
	M_LogEventGeneral('Resetting ADC device...');
ELSIF cmd = E_MA_COMMAND.ENABLE THEN
	pMotor1^.RPC_SetLog(TRUE);
	pMotor2^.RPC_SetLog(TRUE);
	M_SetStatus('');		
	M_LogEventGeneral('Enabling ADC device...');
ELSIF cmd = E_MA_COMMAND.INIT THEN
	pMotor1^.RPC_SetLog(TRUE);
	pMotor2^.RPC_SetLog(TRUE);
	M_SetStatus('Initialising ADC device...');		
	M_LogEventGeneral('Initialising ADC device...');
ELSIF cmd = E_MA_COMMAND.START_TRACK THEN
	pMotor1^.RPC_SetLog(FALSE);
	pMotor2^.RPC_SetLog(FALSE);
	IF mode= E_ADC_MODE.AUTO THEN
		M_SetStatus('Tracking in AUTO mode');
		M_LogEventGeneral('Setting ADC device to AUTO mode...');
	END_IF
ELSIF cmd = E_MA_COMMAND.DISABLE THEN
	M_SetStatus('');		
	M_LogEventGeneral('Disabling ADC device...');
ELSIF cmd = E_MA_COMMAND.STOP THEN
	pMotor1^.RPC_SetLog(TRUE);
	pMotor2^.RPC_SetLog(TRUE);
	M_LogEventGeneral('Stopping ADC device...');
ELSIF cmd = E_MA_COMMAND.STOP_TRACK THEN
	pMotor1^.RPC_SetLog(TRUE);
	pMotor2^.RPC_SetLog(TRUE);
	IF mode= E_ADC_MODE.ENG THEN
		M_SetStatus('Moving to Engineering position ...');		
		M_LogEventGeneral('Setting ADC device to ENGINEERING mode...');
	ELSIF mode= E_ADC_MODE.OFF THEN
		M_SetStatus('Moving to OFF (HOME) position ...');		
		M_LogEventGeneral('Setting ADC device to OFF mode...');
	END_IF
END_IF
END_METHOD

{attribute 'TcRpcEnable':='1'}
METHOD RPC_Disable : INT
VAR_INPUT
END_VAR

VAR 
	i: INT;
END_VAR

// It does all the verifications for the MOTOR device before
// triggering the Disable event.

// RPC calls are not allowed in Local mode.

FOR i := 1 TO nNumAxes DO
	IF ptrMotorStat[i]^.bLocal THEN
		RPC_Disable	:= M_SetRpcStatus(E_MA_RPC_ERROR.LOCAL);
		RETURN;
	END_IF


	// Disable command is accepted only if device is in OP state.
	IF ptrMotorStat[i]^.nState <> E_MOTOR_STATE.OP THEN
		RPC_Disable	:= M_SetRpcStatus(E_MA_RPC_ERROR.NOT_OP);
		RETURN;
		
	END_IF
END_FOR

RefCtrl.nCommand := E_MA_COMMAND.DISABLE;
RefCtrl.bExecute := TRUE;

	
// Call was successful
RPC_Disable	:= M_SetRpcStatus(E_MA_RPC_ERROR.OK);
END_METHOD

{attribute 'TcRpcEnable':='1'}
METHOD RPC_Enable : INT
VAR_INPUT
END_VAR

VAR 
	i: INT;
END_VAR
//
// Check if it is safe to operate motors.
//
IF NOT in_bSafe	THEN
	RPC_Enable	:= M_SetRpcStatus(E_MA_RPC_ERROR.UNSAFE);
	RETURN;
END_IF



// It does all the verifications for the MOTOR device before
// triggering the Enable event.

FOR i := 1 TO nNumAxes DO
	// RPC calls are not allowed in Local mode.
	IF ptrMotorStat[i]^.bLocal THEN
		RPC_Enable	:= M_SetRpcStatus(E_MA_RPC_ERROR.LOCAL);
		RETURN;
	END_IF

	// Enable command is accepted only if device is in NOTOP_READY.
	IF	ptrMotorStat[i]^.nSubstate <> E_MOTOR_SUBSTATE.NOTOP_READY		THEN
		RPC_Enable	:= M_SetRpcStatus(E_MA_RPC_ERROR.NOT_NOTOP_READY);
		RETURN;
	END_IF
END_FOR



// Set enable command
RefCtrl.nCommand := E_MA_COMMAND.ENABLE;
RefCtrl.bExecute := TRUE;
	
// Call was successful
RPC_Enable	:= M_SetRpcStatus(E_MA_RPC_ERROR.OK);
END_METHOD

{attribute 'TcRpcEnable':='1'}
METHOD RPC_Init : INT
VAR_INPUT
END_VAR

VAR 
	i: INT;
END_VAR
M_LogEventGeneral('Initialising ADC motors...');

//
// Check if it is safe to operate motors.
//
IF NOT in_bSafe	THEN
	RPC_Init	:= M_SetRpcStatus(E_MA_RPC_ERROR.UNSAFE);
	RETURN;
END_IF


RPC_Init	:= SUPER^.RPC_Init();
END_METHOD

{attribute 'TcRpcEnable':='1'}
METHOD RPC_MoveAbs : INT
VAR_INPUT
	in_axis:	E_ADC_AXES_ID := E_ADC_AXES_ID.ALL_AXES;
	in_lrPos:	LREAL;
	in_lrVel:	LREAL;
END_VAR

VAR 
	i: INT := 0;
END_VAR
//
// Check if it is safe to operate motors.
//
IF NOT in_bSafe	THEN
	RPC_MoveAbs	:= M_SetRpcStatus(E_MA_RPC_ERROR.UNSAFE);
	RETURN;
END_IF


// Commands are acceptred only when OPERATIONAL
IF	stat.sm.nState <> E_MA_STATE.OP	THEN
	RPC_MoveAbs	:= M_SetRpcStatus(E_MA_RPC_ERROR.NOT_OP);
	RETURN;
// Set velocity cannot be <=0.0.
ELSIF	in_lrVel <= 0.0	THEN
	RPC_MoveAbs	:= M_SetRpcStatus(E_MOTOR_RPC_ERROR.VEL_NEG);
	RETURN;
END_IF

// Check velocity against Vel_max
IF in_axis = E_ADC_AXES_ID.ALL_AXES THEN
	FOR i := 1 TO nNumAxes DO
		// Check if Velocity is too high.
		IF in_lrVel > ptrMotorStat[i]^.axis.lrMaxVelocity THEN
			RPC_MoveAbs	:= M_SetRpcStatus(E_MOTOR_RPC_ERROR.VEL_MAX);
			RETURN;
		END_IF
	END_FOR
ELSE
	// Check if Velocity is too high.
	IF in_lrVel > ptrMotorStat[in_axis]^.axis.lrMaxVelocity THEN
		RPC_MoveAbs	:= M_SetRpcStatus(E_MOTOR_RPC_ERROR.VEL_MAX);
		RETURN;
	END_IF
END_IF


// Set target position
IF in_axis = E_ADC_AXES_ID.ALL_AXES THEN
	FOR i := 1 TO nNumAxes DO
		// RPC calls are not allowed in Local mode.
		IF ptrMotorStat[i]^.bLocal THEN
			RPC_MoveAbs	:= M_SetRpcStatus(E_MA_RPC_ERROR.LOCAL);
			RETURN;
		// Move Absolute command is accepted only in OP state.
		ELSIF	ptrMotorStat[i]^.nState <> E_MOTOR_STATE.OP	THEN
			RPC_MoveAbs	:= M_SetRpcStatus(E_MA_RPC_ERROR.NOT_OP);
			RETURN;
		END_IF
	
		ctrl.lrTargetPos[i] := in_lrPos;
	END_FOR
ELSE
	// RPC calls are not allowed in Local mode.
	IF ptrMotorStat[in_axis]^.bLocal THEN
		RPC_MoveAbs	:= M_SetRpcStatus(E_MA_RPC_ERROR.LOCAL);
		RETURN;
	// Move Absolute command is accepted only in OP state.
	ELSIF	ptrMotorStat[in_axis]^.nState <> E_MOTOR_STATE.OP	THEN
		RPC_MoveAbs	:= M_SetRpcStatus(E_MA_RPC_ERROR.NOT_OP);
		RETURN;
	END_IF
	
	// Ensure moving only one motor
	FOR i := 1 TO nNumAxes DO
		ctrl.lrTargetPos[i] := ptrMotorStat[i]^.lrPosActual;
	END_FOR
	ctrl.lrTargetPos[in_axis] := in_lrPos;
END_IF

SetState(E_MA_STATE.OP, E_MA_SUBSTATE.OP_MOVING);
// Set command
ctrl.lrTargetVel    := in_lrVel;	
ctrl.nCommand 		:= E_MA_COMMAND.MA_MOVE;
ctrl.nMode          := E_ADC_MODE.ENG;
ctrl.bExecute 		:= TRUE;


// Call was successful
RPC_MoveAbs	:= M_SetRpcStatus(E_MA_RPC_ERROR.OK);
END_METHOD

{attribute 'TcRpcEnable':='1'}
METHOD RPC_MoveAngle : INT
VAR_INPUT
	in_lrAngle:	LREAL;
END_VAR

VAR 
	i: INT := 0;
END_VAR
//
// Check if it is safe to operate motors.
//
IF NOT in_bSafe	THEN
	RPC_MoveAngle	:= M_SetRpcStatus(E_MA_RPC_ERROR.UNSAFE);
	RETURN;
END_IF



IF	stat.sm.nState <> E_MA_STATE.OP	THEN
	RPC_MoveAngle	:= M_SetRpcStatus(E_MA_RPC_ERROR.NOT_OP);
	RETURN;
END_IF


FOR i := 1 TO nNumAxes DO
		// RPC calls are not allowed in Local mode.
	IF ptrMotorStat[i]^.bLocal THEN
		RPC_MoveAngle	:= M_SetRpcStatus(E_MA_RPC_ERROR.LOCAL);
		RETURN;
		// Move Absolute command is accepted only in OP state.
	ELSIF	ptrMotorStat[i]^.nState <> E_MOTOR_STATE.OP	THEN
		RPC_MoveAngle	:= M_SetRpcStatus(E_MA_RPC_ERROR.NOT_OP);
		RETURN;
	END_IF
	
	ctrl.lrPosang[i] := in_lrAngle;
END_FOR



SetState(E_MA_STATE.OP, E_MA_SUBSTATE.OP_MOVING);
// Set command
ctrl.nMode:=E_ADC_MODE.OFF;
ctrl.nCommand:= E_MA_COMMAND.STOP_TRACK;
ctrl.bExecute:= TRUE;

// Call was successful
RPC_MoveAngle	:= M_SetRpcStatus(E_MA_RPC_ERROR.OK);
END_METHOD

{attribute 'TcRpcEnable':='1'}
METHOD RPC_MoveRel : INT
VAR_INPUT
	in_axis:	E_ADC_AXES_ID := E_ADC_AXES_ID.ALL_AXES;
	in_lrPos:	LREAL;
	in_lrVel:	LREAL;
END_VAR

VAR 
	i: INT := 0;
	res: INT := E_MOTOR_RPC_ERROR.OK;
END_VAR
//
// Check if it is safe to operate motors.
//
IF NOT in_bSafe	THEN
	RPC_MoveRel	:= M_SetRpcStatus(E_MA_RPC_ERROR.UNSAFE);
	RETURN;
END_IF


// Commands are acceptred only when OPERATIONAL
IF	stat.sm.nState <> E_MA_STATE.OP	THEN
	RPC_MoveRel	:= M_SetRpcStatus(E_MA_RPC_ERROR.NOT_OP);
	RETURN;
// Set velocity cannot be <=0.0.
ELSIF	in_lrVel <= 0.0	THEN
	RPC_MoveRel	:= M_SetRpcStatus(E_MOTOR_RPC_ERROR.VEL_NEG);
	RETURN;
END_IF

// Check velocity against Vel_max
IF in_axis = E_ADC_AXES_ID.ALL_AXES THEN
	FOR i := 1 TO nNumAxes DO
		// Check if Velocity is too high.
		IF in_lrVel > ptrMotorStat[i]^.axis.lrMaxVelocity THEN
			RPC_MoveRel	:= M_SetRpcStatus(E_MOTOR_RPC_ERROR.VEL_MAX);
			RETURN;
		END_IF
	END_FOR
ELSE
	// Check if Velocity is too high.
	IF in_lrVel > ptrMotorStat[in_axis]^.axis.lrMaxVelocity THEN
		RPC_MoveRel	:= M_SetRpcStatus(E_MOTOR_RPC_ERROR.VEL_MAX);
		RETURN;
	END_IF
END_IF


// Set target position
IF in_axis = E_ADC_AXES_ID.ALL_AXES THEN
	FOR i := 1 TO nNumAxes DO
		// RPC calls are not allowed in Local mode.
		IF ptrMotorStat[i]^.bLocal THEN
			RPC_MoveRel	:= M_SetRpcStatus(E_MA_RPC_ERROR.LOCAL);
			RETURN;
		// Move Relative command is accepted only in OP state.
		ELSIF	ptrMotorStat[i]^.nState <> E_MOTOR_STATE.OP	THEN
			RPC_MoveRel	:= M_SetRpcStatus(E_MA_RPC_ERROR.NOT_OP);
			RETURN;
		END_IF
	
		ctrl.lrTargetPos[i] := ptrMotorStat[i]^.lrPosActual + in_lrPos;
	END_FOR
ELSE
	// RPC calls are not allowed in Local mode.
	IF ptrMotorStat[in_axis]^.bLocal THEN
		RPC_MoveRel	:= M_SetRpcStatus(E_MA_RPC_ERROR.LOCAL);
		RETURN;
	// Move Relative command is accepted only in OP state.
	ELSIF	ptrMotorStat[in_axis]^.nState <> E_MOTOR_STATE.OP	THEN
		RPC_MoveRel	:= M_SetRpcStatus(E_MA_RPC_ERROR.NOT_OP);
		RETURN;
	END_IF
	
	// Ensure moving only one motor
	FOR i := 1 TO nNumAxes DO
		ctrl.lrTargetPos[i] := ptrMotorStat[i]^.lrPosActual;
	END_FOR
	ctrl.lrTargetPos[in_axis] := ptrMotorStat[in_axis]^.lrPosActual + in_lrPos;
END_IF

SetState(E_MA_STATE.OP, E_MA_SUBSTATE.OP_MOVING);
// Set command
ctrl.lrTargetVel    := in_lrVel;	
ctrl.nCommand 		:= E_MA_COMMAND.MA_MOVE;
ctrl.nMode          := E_ADC_MODE.ENG;
ctrl.bExecute 		:= TRUE;


// Call was successful
RPC_MoveRel	:= M_SetRpcStatus(E_MA_RPC_ERROR.OK);
END_METHOD

{attribute 'TcRpcEnable':='1'}
METHOD RPC_MoveVel : INT
VAR_INPUT
	in_axis:	E_ADC_AXES_ID := E_ADC_AXES_ID.ALL_AXES;
	in_lrVel:	LREAL;
END_VAR

VAR 
	i: INT := 0;
	res: INT := E_MOTOR_RPC_ERROR.OK;
	dir:	DINT;
END_VAR
//
// Check if it is safe to operate motors.
//
IF NOT in_bSafe	THEN
	RPC_MoveVel	:= M_SetRpcStatus(E_MA_RPC_ERROR.UNSAFE);
	RETURN;
END_IF


IF	stat.sm.nState <> E_MA_STATE.OP	THEN
	RPC_MoveVel	:= M_SetRpcStatus(E_MA_RPC_ERROR.NOT_OP);
	RETURN;
// Set velocity cannot be 0.0.
ELSIF	in_lrVel = 0.0	THEN
	RPC_MoveVel	:= M_SetRpcStatus(E_MOTOR_RPC_ERROR.VEL_ZERO);
	RETURN;
END_IF

// Check velocity against Vel_max.
// Note: Negative velocity is accepted.
IF in_axis = E_ADC_AXES_ID.ALL_AXES THEN
	FOR i := 1 TO nNumAxes DO
		// Check if Velocity is too high.
		IF ABS(in_lrVel) > ptrMotorStat[i]^.axis.lrMaxVelocity THEN
			RPC_MoveVel	:= M_SetRpcStatus(E_MOTOR_RPC_ERROR.VEL_MAX);
			RETURN;
		END_IF
	END_FOR
ELSE
	// Check if Velocity is too high.
	IF ABS(in_lrVel) > ptrMotorStat[in_axis]^.axis.lrMaxVelocity THEN
		RPC_MoveVel	:= M_SetRpcStatus(E_MOTOR_RPC_ERROR.VEL_MAX);
		RETURN;
	END_IF
END_IF

// Update State and Status
SetState(E_MA_STATE.OP, E_MA_SUBSTATE.OP_MOVING);
M_SetStatus('Moving in Velocity mode...');
ctrl.nMode	:= E_ADC_MODE.ENG;

// Set the direction of movement.
IF in_lrVel > 0.0	THEN
	dir	:= MC_Positive_Direction;
ELSE
	dir	:= MC_Negative_Direction;
END_IF


// Restart timer
M_RestartTimer (RefCfg.timeout.nMoveTimeout);

// Command motors to move in velocity.
// This is almost the same as ActionMoveVelExecute().
// Note: Velocity is set with absolute value and direction.
IF in_axis = E_ADC_AXES_ID.ALL_AXES THEN
// Move all axes
	FOR i := 1 TO nNumAxes DO
		ptrMotorCtrl[i]^.nCommand 	:= E_MOTOR_COMMAND.MOTOR_MOVE;
		ptrMotorCtrl[i]^.nMoveType	:= E_MOTOR_MOVE_TYPE.VELOCITY;
		ptrMotorCtrl[i]^.lrVelocity	:= ABS(in_lrVel);
		ptrMotorCtrl[i]^.nDirection	:= dir;
		ptrMotorCtrl[i]^.bExecute	:= TRUE;
	END_FOR
ELSE
// Move only the selected axis
	ptrMotorCtrl[in_axis]^.nCommand 	:= E_MOTOR_COMMAND.MOTOR_MOVE;
	ptrMotorCtrl[in_axis]^.nMoveType	:= E_MOTOR_MOVE_TYPE.VELOCITY;
	ptrMotorCtrl[in_axis]^.lrVelocity	:= ABS(in_lrVel);
	ptrMotorCtrl[in_axis]^.nDirection	:= dir;
	ptrMotorCtrl[in_axis]^.bExecute		:= TRUE;
END_IF



// Call was successful
RPC_MoveVel	:= M_SetRpcStatus(E_MA_RPC_ERROR.OK);
END_METHOD

{attribute 'TcRpcEnable':='1'}
METHOD RPC_Reset : INT
VAR_INPUT
END_VAR

VAR 
	i: INT;
END_VAR

FOR i := 1 TO nNumAxes DO
	// RPC calls are not allowed in Local mode.
	IF ptrMotorStat[i]^.bLocal THEN
		RPC_Reset	:= M_SetRpcStatus(E_MA_RPC_ERROR.LOCAL);
		RETURN;
	END_IF
END_FOR


ctrl.nCommand := E_MA_COMMAND.RESET;
ctrl.bExecute := TRUE;

// Call was successful
RPC_Reset	:= M_SetRpcStatus(E_MA_RPC_ERROR.OK);
END_METHOD

{attribute 'TcRpcEnable':='1'}
METHOD RPC_StartTrack : INT
VAR_INPUT
	in_angle:    LREAL := 0.0;
END_VAR

VAR 
	i: INT;
END_VAR
//
// Check if it is safe to operate motors.
//
IF NOT in_bSafe	THEN
	RPC_StartTrack	:= M_SetRpcStatus(E_MA_RPC_ERROR.UNSAFE);
	RETURN;
END_IF



FOR i := 1 TO nNumAxes DO
	// RPC calls are not allowed in Local mode.
	IF ptrMotorStat[i]^.bLocal THEN
		RPC_StartTrack	:= M_SetRpcStatus(E_MA_RPC_ERROR.LOCAL);
		RETURN;
	// Move Absolute command is accepted only in OP state.
	ELSIF	ptrMotorStat[i]^.nState <> E_MOTOR_STATE.OP	THEN
		RPC_StartTrack	:= M_SetRpcStatus(E_MA_RPC_ERROR.NOT_OP);
		RETURN;
	END_IF
END_FOR


// Set command
ctrl.lrPosang[1] := in_angle;
ctrl.lrPosang[2] := in_angle;

ctrl.nMode:= E_ADC_MODE.AUTO;
ctrl.nCommand:=E_MA_COMMAND.START_TRACK;
ctrl.bExecute:=(TRUE);

// Call was successful
RPC_StartTrack	:= M_SetRpcStatus(E_MA_RPC_ERROR.OK);
END_METHOD

{attribute 'TcRpcEnable':='1'}
METHOD RPC_Stop : INT
VAR_INPUT
END_VAR

VAR 
	i: INT;
END_VAR

FOR i := 1 TO nNumAxes DO
	// RPC calls are not allowed in Local mode.
	IF ptrMotorStat[i]^.bLocal THEN
		RPC_Stop	:= M_SetRpcStatus(E_MA_RPC_ERROR.LOCAL);
		RETURN;
	END_IF
END_FOR



ctrl.nCommand := E_MA_COMMAND.STOP;
ctrl.bExecute := TRUE;

RPC_Stop	:= M_SetRpcStatus(E_MA_RPC_ERROR.OK);
END_METHOD

{attribute 'TcRpcEnable':='1'}
METHOD RPC_StopTrack : INT
VAR_INPUT
END_VAR

VAR 
	i: INT;
END_VAR

IF (RefStat.nMode = E_ADC_MODE.AUTO) THEN
	FOR i := 1 TO nNumAxes DO
		// RPC calls are not allowed in Local mode.
		IF ptrMotorStat[i]^.bLocal THEN
			RPC_StopTrack	:= M_SetRpcStatus(E_MA_RPC_ERROR.LOCAL);
			RETURN;
		END_IF
	END_FOR

	SetState(E_MA_STATE.OP, E_MA_SUBSTATE.OP_MOVING);
	RefCtrl.nMode           :=  E_ADC_MODE.OFF;
	// Set command
	RefCtrl.nCommand 		:= E_MA_COMMAND.STOP_TRACK;
	RefCtrl.bExecute 		:= TRUE;
END_IF

// Call was successful
RPC_StopTrack	:= M_SetRpcStatus(E_MA_RPC_ERROR.OK);
END_METHOD

METHOD User_ComputeAutoPos : LREAL
VAR_INPUT
	index:	INT;	// ADC index [1..2]
END_VAR

VAR
	pos_deg:		LREAL := 0.0;
	adcPos:	    	LREAL := 0.0;
	latitude:       LREAL := stSiteConstants.latitude;
	adaPosang:	    LREAL := stat.lrAdaPosAngle  * GCL.C_DEG2RAD;	// TODO: check
	drotPos:		LREAL := stat.lrDrotPos * GCL.C_DEG2RAD;
	ra:             LREAL := stPointingKernel.radec_at_altaz_at_requested_xy[0];
	dec:            LREAL := stPointingKernel.radec_at_altaz_at_requested_xy[1];
	pressure:       LREAL := stEnvironmentData.pressure;
	temperature:    LREAL := stEnvironmentData.temperature;
	ha:             LREAL ;
	alt:            LREAL := stPointingKernel.target_observed_altaz[0];
	pa:		    	LREAL;	// Parallactic angle [rad]
	cos_pa:			LREAL;
	sin_pa:			LREAL;
    zd:             LREAL := 0.0;   // zenith distance
	rho:			LREAL := 0.0;	// Parallactic Angle component
	phi:			LREAL := 0.0;	// Refraction component

	C:				LREAL := 0.0;	// Total Correction = CO + CP + CT
	CO:				LREAL := 0.0;	// Correction for Offset
	CP:				LREAL := 0.0;	// Correction for Pressure
	CT:				LREAL := 0.0;	// Correction for Temperature
	tempVar:		LREAL := 0.0;
	
	posOffset:	    LREAL := cfg.unitCfg[index].lrPosOffset * GCL.C_DEG2RAD;
	minElev:		LREAL := cfg.lrMinElev   * GCL.C_DEG2RAD;
	
END_VAR

// FOR elev > 27.64:
// A = C * tan(zd)
// zd = 90 - elev
// C = CO + CP + CT
// CO = Coffset = 1.7387
// CP = Pslope * (P - Poffset) = 0.0023 * (P - 743)
// CT = Tslope * (T - Toffset) = -0.0061 * (T - 12)

ha := stPointingKernel.time_lst - ra;
zd := GCL.C_PI2 - stPointingKernel.target_observed_altaz[0];		// Zenith distance = PI/2 - Alt
// Select DROT or ADA position based on the DROT factor
IF (ABS(cfg.unitCfg[index].lrDrotFactor) <> 2) THEN	
			drotPos := adaPosang;
END_IF			

// Calculate the parallactic angle				
IF (zd <= cfg.lrZDlimit) THEN
			// If we are too close to Zenith, set parallactic angle to zero
			pa := 0.0;
ELSE
	IF ((COS(dec) * SIN(zd) = 0.0)) THEN
		cos_pa := 0.0;
	ELSE
		cos_pa := (SIN(latitude) - SIN(dec) * COS(zd)) / (COS(dec) * SIN(zd));
	END_IF
	IF (SIN(zd) = 0.0) THEN
		sin_pa := 0.0;
	ELSE
		sin_pa := (COS(latitude) * SIN(ha)) / SIN(zd);
	END_IF
			
	IF (cos_pa >= 0) THEN
		pa := ASIN(sin_pa);
	ELSE
		pa := GCL.C_PI - ASIN(sin_pa);
    END_IF
END_IF
		
//
// Calculate corrections
// rho = nominal ADC position without corrections
//
// TODO: This seems to be overwritten?
// This might be the right formula !!!
rho := posOffset - adaPosang - pa;
		
IF (alt <= minElev) THEN
	// No corrections for altitudes below minimum elevation	
	rho := posOffset + minElev + cfg.unitCfg[index].lrDrotFactor * drotPos;
	adcPos := rho;					
ELSE
    rho := posOffset + alt + cfg.unitCfg[index].lrDrotFactor * drotPos;
	// TODO: NOTE: This might be just rho := posOffset_r - pa
	// Talk to Joel.
			
	// Correction for Offset
	CO := cfg.unitCfg[index].lrCoffset;
			
	// Correction for Pressure.
	IF	pressure >= GCL.C_MIN_P AND pressure <= GCL.C_MAX_P	THEN
		// Correct for Pressure only if pressure offset is defined
		IF (cfg.lrPoffset <> 0.0) THEN
					CP := cfg.lrPslope * (pressure - cfg.lrPoffset);
		END_IF			
	END_IF

	// Correction for Temperature?
	IF	temperature >= GCL.C_MIN_T AND temperature <= GCL.C_MAX_T	THEN
		// Correct for Temperature only if temperature offset is defined
		IF (cfg.lrToffset <> 0.0) THEN
			CT := cfg.lrTslope * (temperature - cfg.lrToffset);
		END_IF			
	END_IF

	// TODO: Humidity effect correction?
			
	// Total correction
	C := CO + CP + CT;
			
	// Altitude effect correction only if within limits
	// tempVar := GCL.C_PI2 - alt_r;	// TODO: Removed
	IF ((alt <= 0) OR (alt >= GCL.C_2PI)) THEN
		tempVar := 0;
	ELSE
		tempVar := TAN(GCL.C_PI2 - alt);
	END_IF
			
	IF (cfg.lrAfactor = 0.0) THEN
		tempVar := 0;	// No compensation!
	ELSE
		tempVar := C * tempVar / cfg.lrAfactor;
	END_IF
			
			
	// tempVar is a COS(), i.e. must be ABS(tempVar) < 1.0
	IF (ABS(tempVar) >= 1.0) THEN
		phi := 0;
	ELSE
		phi := ACOS(tempVar);
	END_IF		
		adcPos := rho + (cfg.unitCfg[index].nSignPhi * phi);					
END_IF	
		
pos_deg := cfg.unitCfg[index].lrRefAuto + (cfg.unitCfg[index].nSignAuto * adcPos * GCL.C_RAD2DEG);

User_ComputeAutoPos := pos_deg;
END_METHOD

METHOD User_ComputeNextPos : BOOL
VAR_INPUT
END_VAR
VAR
	i:	INT;
	pos_deg:		LREAL := 0.0;
END_VAR

FOR i := 1 TO nNumAxes DO
	
// Handle various ADC modes
// Set both position and velocity depending on the mode.
//
// Position [deg]
// Velocity [deg/sec]:
//    ENG  - as given in adcCtrl.lrTargetVel
//    OFF  - default motor velocity
//    AUTO - default motor velocity
	CASE RefStat.nMode OF
		E_ADC_MODE.ENG:	// MULTI_MODE_ENG
			pos_deg:= ctrl.lrTargetPos[i];
			
			ptrMotorCtrl[i]^.lrVelocity := ctrl.lrTargetVel;		
			M_SetStatus('Moving to Engineering position ...');
		E_ADC_MODE.OFF:	// MULTI_MODE_1
			// TODO: Say why POSANG + REF OFFSET
			//       The motor should go to 0.0, i.e. HOME?
			pos_deg := cfg.unitCfg[i].lrRefOff + cfg.unitCfg[i].nSignOff * (ctrl.lrPosang[i]); // computation in degrees
			ptrMotorCtrl[i]^.lrVelocity := ptrMotorCfg[i]^.lrDefaultVelocity;		
			M_SetStatus('Homing motors ...');
		E_ADC_MODE.AUTO:	// MULTI_MODE_2
			pos_deg := User_ComputeAutoPos(i);
			ptrMotorCtrl[i]^.lrVelocity := ptrMotorCfg[i]^.lrDefaultVelocity;
			M_SetStatus('Moving in AUTO mode ...');
	END_CASE
	// assign new position
	ptrMotorCtrl[i]^.lrPosition := pos_deg;
END_FOR


User_ComputeNextPos := TRUE;
END_METHOD

// Method for hard-coding of configuration parameters by the User.
METHOD User_Configure : BOOL
VAR_INPUT
END_VAR
SUPER^.User_Configure();	// Mandatory!

//
// TODOUSER: Configure anything that is different from default configuration.
//
// Examples:
//
// ADC configuration
cfg.unitCfg[1].nSignOff	:=  1;
cfg.unitCfg[2].nSignOff	:=  1;

cfg.unitCfg[1].nSignPhi	:=  1;
cfg.unitCfg[2].nSignPhi	:= -1;

//
// Individual Motor configuration
ptrMotorCfg[1]^.nAxisType	:= E_MOTOR_AXIS_TYPE.CIRCULAR_OPTIMISED;
ptrMotorCfg[2]^.nAxisType	:= E_MOTOR_AXIS_TYPE.CIRCULAR_OPTIMISED;

ptrMotorCfg[1]^.lrDefaultVelocity	:= 10.0;	// Set default velocity to 10 deg/sec
ptrMotorCfg[2]^.lrDefaultVelocity	:= 10.0;	// Set default velocity to 10 deg/sec

// Multi-axis system configuration
ctrl.lrPosang[1]	:=  0.0;	// Position angle for OFF mode, i.e. HOME position
ctrl.lrPosang[2]	:=  0.0;	// Position angle for OFF mode, i.e. HOME position
ctrl.lrTargetPos[1]	:= 45.0;	// ADC1 Position angle for ENG mode
ctrl.lrTargetPos[2]	:= 45.0;	// ADC2 Position angle for ENG mode
ctrl.lrTargetVel	:= 10.0;	// Velocity for ENG mode
END_METHOD

// User Method executed on each cycle before processing events and states.
METHOD User_GetParams : BOOL
VAR_INPUT
END_VAR
VAR
	i:	INT;
END_VAR
//
// TODOUSER: Set anything that should be set on every cycle, if any.
//
//
SUPER^.User_GetParams();

// Example: Any settings that are mode dependant.
CASE RefCtrl.nMode OF
			MA_MODE_ENG:
			    ; 
END_CASE
END_METHOD

// User Method executed on each cycle after processing events and states.
METHOD User_SetParams : BOOL
VAR_INPUT
END_VAR
VAR
	i:		INT;
END_VAR
//
// Mandatory
//
SUPER^.User_SetParams();

// Set maximum positioning error
stat.lrPosError		:= M_GetMaxPosError();

// Check if we are tracking or still presetting.
// Tracking is OK if the positioning error is less than the threshold (bTrackingOK).
// Once device is tracking, it should go back to presetting if the error is greater
// than twice the threshold  (bTrackingBAD).
IF ctrl.nMode = E_ADC_MODE.AUTO THEN
	stat.bTrackingOK	:= SEL (stat.lrPosError <= cfg.lrTrkThreshold, FALSE, TRUE);
	stat.bTrackingBAD	:= SEL (stat.lrPosError > 2.0 * cfg.lrTrkThreshold, FALSE, TRUE);
	stat.lrAlt := stPointingKernel.target_observed_altaz[0] * GCL.C_RAD2DEG;
    stat.lrAz := stPointingKernel.target_observed_altaz[1] * GCL.C_RAD2DEG;
	stat.lrRa := F_astroRad2Hms(stPointingKernel.radec_at_altaz_at_requested_xy[0]);
	stat.lrDec := F_astroRad2Dms(stPointingKernel.radec_at_altaz_at_requested_xy[1]);
	stat.lrPa := stPointingKernel.parallactic_angle * GCL.C_RAD2DEG;
ELSE
	stat.bTrackingOK	:= FALSE;
	stat.bTrackingBAD	:= FALSE;
END_IF
END_METHOD

END_FUNCTION_BLOCK

// ---- POUs/MultiAxis/FB_MA_BASE.TcPOU
FUNCTION_BLOCK FB_MA_BASE
VAR_INPUT
	{attribute 'OPC.UA.DA' := '0'}
	sName:			STRING	:= 'MA';	// Default system name, e.g. 'ADC'
	{attribute 'OPC.UA.DA' := '0'}
	nNumAxes:		INT		:= 1;		// Total number of motors/axes, max 6
	// Pointers to motors.
	// It must be at least two motors, so no defaults to zero for the first two.
	{attribute 'OPC.UA.DA' := '0'}
	pMotor1:		POINTER TO FB_MOTOR;
	{attribute 'OPC.UA.DA' := '0'}
	pMotor2:		POINTER TO FB_MOTOR	:= 0;
	{attribute 'OPC.UA.DA' := '0'}
	pMotor3:		POINTER TO FB_MOTOR	:= 0;
	{attribute 'OPC.UA.DA' := '0'}
	pMotor4:		POINTER TO FB_MOTOR	:= 0;
	{attribute 'OPC.UA.DA' := '0'}
	pMotor5:		POINTER TO FB_MOTOR	:= 0;
	{attribute 'OPC.UA.DA' := '0'}
	pMotor6:		POINTER TO FB_MOTOR	:= 0;

	// EICSSW-1923
	{attribute 'OPC.UA.DA' := '0'}
	in_bSafe:		BOOL	:= TRUE;	// Flag if safe to move the motor
	{attribute 'OPC.UA.DA' := '0'}
	in_bDisableIfUnsafe:	BOOL := FALSE;	// If unsafe, motor is disabled
END_VAR
VAR
	
	// Pointers to motors configuration, control and status.
	// Initialised in M_Configure().
	{attribute 'OPC.UA.DA' := '0'}
	pMotor:			ARRAY [1..GPL.C_MA_MAX_AXES] OF POINTER TO FB_MOTOR;
	{attribute 'OPC.UA.DA' := '0'}
	ptrMotorCfg:	ARRAY [1..GPL.C_MA_MAX_AXES] OF POINTER TO T_MOTOR_CFG;
	{attribute 'OPC.UA.DA' := '0'}
	ptrMotorCtrl:	ARRAY [1..GPL.C_MA_MAX_AXES] OF POINTER TO T_MOTOR_CTRL;
	{attribute 'OPC.UA.DA' := '0'}
	ptrMotorStat:	ARRAY [1..GPL.C_MA_MAX_AXES] OF POINTER TO T_MOTOR_STAT;
	
	// References
	{attribute 'OPC.UA.DA' := '0'}
	RefCfg:			REFERENCE TO T_MA_CFG;	    // Reference to Config parameters
	{attribute 'OPC.UA.DA' := '0'}
	RefCtrl:		REFERENCE TO T_MA_CTRL;	    // Reference to Control parameters
	{attribute 'OPC.UA.DA' := '0'}
	RefStat:		REFERENCE TO T_MA_STAT;	    // Reference to Status parameters

	{attribute 'OPC.UA.DA' := '0'}
	nPtpOffset:   	DINT := 0;			// TODO What is this?
	
	{attribute 'OPC.UA.DA' := '0'}
	nState:       	DINT := E_MA_STATE.NOTOP;
	{attribute 'OPC.UA.DA' := '0'}
	nSubState:    	DINT := E_MA_SUBSTATE.NOTOP_NOTREADY;
	{attribute 'OPC.UA.DA' := '0'}
	sState:			STRING := 'UNKNOWN';
	
	{attribute 'OPC.UA.DA' := '0'}
	nEvent:		      	DINT := E_MA_EVENT.NONE;
	{attribute 'OPC.UA.DA' := '0'}
	nInternalEvent:		DINT := E_MA_EVENT.NONE;

	{attribute 'OPC.UA.DA' := '0'}
	waitTout:     	TON;                    (* General Timeout *)
	
	// Operational Events
	{attribute 'OPC.UA.DA' := '0'}
	fbEventGeneral:	FB_TcMessage;
	{attribute 'OPC.UA.DA' := '0'}
	fbEventError:	FB_TcMessage;
	
END_VAR

// Configure the system, i.e. set pointers
M_Configure();

// If the pointers to motors have not been configured, don't do anything.
// Otherwise the system will crash with exception.
IF NOT RefStat.bConfigured THEN
	RETURN;
END_IF

// Read configuration parameters of the ADC device

//ptrMotorCfg := ADR(motor.cfg);
// Create an instance of the motor device. Internally it handles the axis
//ptrMotorCfg^.nTypeAxis := nAxisType;

// Transfer external parameters to the FB variables.
THIS^.User_GetParams();

// Handles commands received through the external interface, normally OPC-UA.
//THIS^.User_HandleExternalCmds();


// Handles the internal states of the device.
//THIS^.HandleStates();

(* === Check for commands and internal events to be processed === *)
CheckForEvents();

(* === Process events according to the State Machine === *)
ProcessEvents();

// Update device status object
THIS^.User_SetParams();

METHOD ActionDisableExecute 
VAR_INPUT
END_VAR
VAR
	i:		INT;
END_VAR
// Restart timer
M_RestartTimer (RefCfg.timeout.nStopTimeout);

FOR i := 1 TO nNumAxes DO
	// Send DISABLE command to the motors
	ptrMotorCtrl[i]^.nCommand := E_MOTOR_COMMAND.DISABLE;
	ptrMotorCtrl[i]^.bExecute	:= TRUE;
END_FOR
END_METHOD

METHOD ActionEnableExecute 
VAR_INPUT
END_VAR
VAR
	i:		INT;
END_VAR
// Restart timer
M_RestartTimer (RefCfg.timeout.nStopTimeout);

FOR i := 1 TO nNumAxes DO
	// Send ENABLE command to the motors
	ptrMotorCtrl[i]^.nCommand := E_MOTOR_COMMAND.ENABLE;
	ptrMotorCtrl[i]^.bExecute	:= TRUE;
END_FOR
END_METHOD

METHOD ActionInitExecute
VAR_INPUT
END_VAR
VAR
	i:		INT;
END_VAR
SetAction('ActionInitExecute');

// Don't move if not safe.
IF (NOT in_bSafe) THEN
	THIS^.M_SetStatus('ERROR: MA cannot INIT. Not safe to move.');
	SetState(E_MA_STATE.NOTOP, E_MA_SUBSTATE.NOTOP_ERROR);
	RETURN;
END_IF




// Restart timer
M_RestartTimer (RefCfg.timeout.nInitTimeout);

// Initialise motors that are NOTOP.
// Motors that are OP_STANDSTILL will be disabled.
// Motors that are moving will be stopped BUT global INIT will fail
// since the system will not end up in NOTOP/READY.
//
FOR i := 1 TO nNumAxes DO
	IF	ptrMotorStat[i]^.nState = E_MOTOR_STATE.NOTOP	THEN
		ptrMotorCtrl[i]^.nCommand := E_MOTOR_COMMAND.INIT;
	ELSIF ptrMotorStat[i]^.nSubstate = E_MOTOR_SUBSTATE.OP_STANDSTILL THEN
		ptrMotorCtrl[i]^.nCommand := E_MOTOR_COMMAND.DISABLE;
	ELSE
		// Motor will stop but INIT will fail with timeout!!!
		ptrMotorCtrl[i]^.nCommand := E_MOTOR_COMMAND.STOP;
	END_IF

	// Execute the commands
	ptrMotorCtrl[i]^.bExecute	:= TRUE;
END_FOR

// Set NOT Initialised
M_SetInit(FALSE);
END_METHOD

// Move motors. Pos and Vel are already set!
METHOD ActionMoveAbsExecute
VAR_INPUT
END_VAR
VAR
	i:			INT;
END_VAR
// Restart timer
M_RestartTimer (RefCfg.timeout.nMoveTimeout);

// Move all axis.
// Pos and Vel are already set!
FOR i := 1 TO nNumAxes DO
	ptrMotorCtrl[i]^.nCommand 	:= E_MOTOR_COMMAND.MOTOR_MOVE;
	ptrMotorCtrl[i]^.nMoveType	:= E_MOTOR_MOVE_TYPE.ABSOLUTE;
	ptrMotorCtrl[i]^.bExecute	:= TRUE;
END_FOR
END_METHOD

METHOD ActionMoveVelExecute
VAR_INPUT
	vel: LREAL;
    dir: DINT;
END_VAR
VAR
	i:		INT;
END_VAR
// Restart timer
M_RestartTimer (RefCfg.timeout.nMoveTimeout);

FOR i := 1 TO nNumAxes DO
	ptrMotorCtrl[i]^.nCommand 	:= E_MOTOR_COMMAND.MOTOR_MOVE;
	ptrMotorCtrl[i]^.nMoveType	:= E_MOTOR_MOVE_TYPE.VELOCITY;
	ptrMotorCtrl[i]^.lrVelocity	:= vel;
	ptrMotorCtrl[i]^.nDirection	:= dir;
	ptrMotorCtrl[i]^.bExecute	:= TRUE;
END_FOR
END_METHOD

METHOD ActionResetExecute 
VAR_INPUT
END_VAR
VAR
	i:		INT;
END_VAR
// Restart timer
M_RestartTimer (RefCfg.timeout.nStopTimeout);

// Send RESET command to the motors
FOR i := 1 TO nNumAxes DO
	ptrMotorCtrl[i]^.nCommand := E_MOTOR_COMMAND.RESET;
	ptrMotorCtrl[i]^.bExecute	:= TRUE;
END_FOR

// Set NOT Initialised
M_SetInit(FALSE);
END_METHOD

METHOD ActionStopExecute
VAR_INPUT
END_VAR
VAR
	i:		INT;
END_VAR
M_SetStatus('Stopping ...');

// Restart timer
M_RestartTimer (RefCfg.timeout.nStopTimeout);

FOR i := 1 TO nNumAxes DO
	// Send STOP command to the motors
	ptrMotorCtrl[i]^.nCommand := E_MOTOR_COMMAND.STOP;
	ptrMotorCtrl[i]^.bExecute	:= TRUE;
END_FOR
END_METHOD

// Move motors in tracking mode. Pos and Vel are already set!
// In tracking mode motor logs are disabled.
// Otherwise the system would be flooded with logs.
METHOD ActionTrackExecute
VAR_INPUT
END_VAR
VAR
	i:			INT;
END_VAR
// Restart timer
M_RestartTimer (RefCfg.timeout.nMoveTimeout);

// Move all axis.
// Pos and Vel are already set!
// Set TRACKING MODE E_MOTOR_MOVE_TYPE.TRACKING !!!
FOR i := 1 TO nNumAxes DO
	ptrMotorCtrl[i]^.nCommand 	:= E_MOTOR_COMMAND.MOTOR_MOVE;
	ptrMotorCtrl[i]^.nMoveType	:= E_MOTOR_MOVE_TYPE.TRACKING;
	ptrMotorCtrl[i]^.bExecute	:= TRUE;
END_FOR
END_METHOD

METHOD ActivityDisabling : BOOL
VAR_INPUT
END_VAR
waitTout (IN := TRUE);	// Update timeout timer

IF M_CheckAxesState(E_MOTOR_STATE.NOTOP, 
					E_MOTOR_SUBSTATE.NOTOP_READY) THEN
	waitTout (IN := FALSE);	// Stop the timer
	SetState(E_MA_STATE.NOTOP, E_MA_SUBSTATE.NOTOP_READY);
	THIS^.M_SetStatus('Motors Disabled');
	RETURN;
END_IF

// Check the timeout
IF waitTout.Q THEN
	waitTout (IN := FALSE);	// Stop the timer
	// Stop the motor
	THIS^.ActionStopExecute();
	THIS^.M_SetStatus('ERROR: Timeout on Disable');
	SetState(E_MA_STATE.NOTOP, E_MA_SUBSTATE.NOTOP_ERROR);
	RETURN;
END_IF
END_METHOD

METHOD ActivityEnabling : BOOL
VAR_INPUT
END_VAR
waitTout (IN := TRUE);	// Update timeout timer

IF M_CheckAxesState(E_MOTOR_STATE.OP, 
					E_MOTOR_SUBSTATE.OP_STANDSTILL) THEN
	waitTout (IN := FALSE);	// Stop the timer
	SetState(E_MA_STATE.OP, E_MA_SUBSTATE.OP_STANDSTILL);
	THIS^.M_SetStatus('Motors Operational');
	RETURN;
END_IF

// Check the timeout
IF waitTout.Q THEN
	waitTout (IN := FALSE);	// Stop the timer
	// Stop the motor
	THIS^.ActionStopExecute();
	THIS^.M_SetStatus('ERROR: Timeout on Enable');
	SetState(E_MA_STATE.NOTOP, E_MA_SUBSTATE.NOTOP_ERROR);
	RETURN;
END_IF
END_METHOD

METHOD ActivityInitialising : BOOL
VAR_INPUT
END_VAR

VAR
END_VAR
(* 
	Activity monitors the MA initialisation task 
*)


SetAction('ActivityInitialising');

waitTout (IN := TRUE);	// Update timeout timer

IF (NOT in_bSafe) THEN
	waitTout (IN := FALSE);	// Stop the timer
	THIS^.M_SetStatus('ERROR: MA error during INIT. Not safe to move.');
	SetState(E_MA_STATE.NOTOP, E_MA_SUBSTATE.NOTOP_ERROR);
	RETURN;
END_IF




IF (M_CheckError()) THEN
	waitTout (IN := FALSE);	// Stop the timer
	THIS^.M_SetStatus('ERROR: MA error during INIT');
	SetState(E_MA_STATE.NOTOP, E_MA_SUBSTATE.NOTOP_ERROR);
	RETURN;
END_IF



//
// The device is initialised if:
// - Motor is initialised, i.e NOTOP_READY
// - The reading of the Leap Second is complete, i.e. bCoEReadFlag = FALSE (if used)
//
IF M_CheckAxesState(E_MOTOR_STATE.NOTOP, 
					E_MOTOR_SUBSTATE.NOTOP_READY) THEN
	waitTout (IN := FALSE);	// Stop the timer
	THIS^.M_SetStatus('Device initialised');
	M_SetInit(TRUE);
	SetState(E_MA_STATE.NOTOP, E_MA_SUBSTATE.NOTOP_READY);
	RETURN;
END_IF

// Check the timeout
IF waitTout.Q THEN
	waitTout (IN := FALSE);	// Stop the timer
	// Stop the motor
	THIS^.ActionStopExecute();
	THIS^.M_SetStatus('ERROR: INIT Timeout!');
	//nInternalEvent  := E_MA_EVENT.ERRINIT;
	SetState(E_MA_STATE.NOTOP, E_MA_SUBSTATE.NOTOP_ERROR);
	RETURN;
END_IF
END_METHOD

METHOD ActivityMoving : BOOL
VAR_INPUT
END_VAR
VAR
	i:		INT;
END_VAR
// If nSkipCycle < GPL.C_CYCLE_IDLE, the motor has not moved off yet.
// Wait GPL.C_CYCLE_IDLE cycles so the motor status has been updated.
//RefStat.nSkippedCycles	:= RefStat.nSkippedCycles + 1;
IF RefStat.nSkippedCycles < RefCfg.nMinSkipCycles THEN
	RETURN;
END_IF

waitTout (IN := TRUE);	// Update timeout timer

// Check for motor errors
IF (M_CheckError()) THEN
	waitTout (IN := FALSE);	// Stop the timer
	RefStat.sStatus	:= 'ERROR: Motor in error state';
	SetState(E_MA_STATE.OP, E_MA_SUBSTATE.OP_ERROR);	
	RETURN;
END_IF

// Check if the motor state is standstill for all motors.
// If yes, the motion is complete.
// Start checking it GPL.C_CYCLE_IDLE after the motor has received the MOVE command.
// EICSSW-706: Also check the positioning error.
IF RefStat.nSkippedCycles > 2*RefCfg.nMinSkipCycles THEN
	// Don't check the status immediately since motor starts from standstill.
	// The timer should have at least one increment, i.e. ET>0.
	IF 	waitTout.ET > INT_TO_TIME(0)							AND
		M_GetMaxPosError() < RefCfg.lrTrkThreshold	AND 
		M_CheckAxesState(E_MOTOR_STATE.OP, 
						 E_MOTOR_SUBSTATE.OP_STANDSTILL)	THEN
		waitTout (IN := FALSE);	// Stop the timer
		SetState(E_MA_STATE.OP, E_MA_SUBSTATE.OP_STANDSTILL);
		THIS^.M_SetStatus('Motors Standstill');
		RETURN;
	END_IF
END_IF


// Check for timeout
IF waitTout.Q THEN
	waitTout (IN := FALSE);	// Stop the timer
	// Stop the motor
	THIS^.ActionStopExecute();
	THIS^.M_SetStatus('ERROR: Motion Timeout');
	SetState(E_MA_STATE.OP, E_MA_SUBSTATE.OP_ERROR);
	RETURN;
END_IF
END_METHOD

METHOD ActivityPresetting : BOOL
VAR_INPUT
END_VAR
// Essentially, Presetting is identical to Tracking with the only difference
// that the actual position is far away from the target position.
ActivityTracking();
END_METHOD

METHOD ActivityResetting : BOOL
VAR_INPUT
END_VAR
waitTout (IN := TRUE);	// Update timeout timer

IF M_CheckAxesState(E_MOTOR_STATE.NOTOP, 
					E_MOTOR_SUBSTATE.NOTOP_NOTREADY) THEN
	SetState(E_MA_STATE.NOTOP, E_MA_SUBSTATE.NOTOP_NOTREADY);
	THIS^.M_SetStatus('Control Reset');
	waitTout (IN := FALSE);	// Stop the timer
	RETURN;
END_IF

// Check the timeout
IF waitTout.Q THEN
	// Stop the motor
	THIS^.ActionStopExecute();
	waitTout (IN := FALSE);	// Stop the timer
	THIS^.M_SetStatus('ERROR: Timeout on Reset');
	SetState(E_MA_STATE.NOTOP, E_MA_SUBSTATE.NOTOP_ERROR);
	RETURN;
END_IF
END_METHOD

METHOD ActivityStopping : BOOL
VAR_INPUT
END_VAR
waitTout (IN := TRUE);	// Update timeout timer

CASE RefStat.sm.nState OF	
	
  E_MA_STATE.NOTOP:	
	//
	// NotOperational - NotRead case
	//
	IF NOT M_CheckAxesState(E_MOTOR_STATE.NOTOP, 
							E_MOTOR_SUBSTATE.NOTOP_INITIALIZING)  THEN
		// If INIT was interrupted, set substate to NOT READY.
		// Otherwise, keep the same state.
		IF M_AxesInitialised() THEN
			SetState(E_MA_STATE.NOTOP, E_MA_SUBSTATE.NOTOP_READY);
		ELSE
			SetState(E_MA_STATE.NOTOP, E_MA_SUBSTATE.NOTOP_NOTREADY);
		END_IF
		THIS^.M_SetStatus('Motors Standstill');
		waitTout (IN := FALSE);	// Stop the timer
		RETURN;
	END_IF

	// Check the timeout
	IF waitTout.Q THEN
		// Stop the motor
		THIS^.ActionStopExecute();
		waitTout (IN := FALSE);	// Stop the timer
		THIS^.M_SetStatus('ERROR: Motors initialization timeout');
		SetState(E_MA_STATE.NOTOP, E_MA_SUBSTATE.NOTOP_ERROR);
		RETURN;
	END_IF

  E_MA_STATE.OP:
	//
	// OPERATIONAL
	//
	IF M_CheckAxesState(E_MOTOR_STATE.OP, 
						E_MOTOR_SUBSTATE.OP_STANDSTILL)  THEN
		SetState(E_MA_STATE.OP, E_MA_SUBSTATE.OP_STANDSTILL);
		THIS^.M_SetStatus('Motors Standstill');
		waitTout (IN := FALSE);	// Stop the timer
		RETURN;
	END_IF

	// Check the timeout
	IF waitTout.Q THEN
		// Stop the motor
		THIS^.ActionStopExecute();
		waitTout (IN := FALSE);	// Stop the timer
		THIS^.M_SetStatus('ERROR: Timeout while stopping motors');
		SetState(E_MA_STATE.OP, E_MA_SUBSTATE.OP_ERROR);
		RETURN;
	END_IF
END_CASE
END_METHOD

METHOD ActivityTracking : BOOL
VAR_INPUT
END_VAR
IF NOT in_bSafe THEN
	RefStat.sStatus	:= 'ERROR: Not safe to move motor.';
	M_LogEventError('Not safe to move motor. Tracking stopped.');	
	SetState(E_MA_STATE.OP, E_MA_SUBSTATE.OP_ERROR);
	RETURN;
END_IF

IF (M_CheckError()) THEN
	RefStat.sStatus	:= 'ERROR: Aborted tracking mode.';
	M_LogEventError('Aborted tracking mode.');	
	SetState(E_MA_STATE.OP, E_MA_SUBSTATE.OP_ERROR);	
	RETURN;
END_IF


// Since it takes at least 4 cycles for a move, new Move command is sent every nCyclesIdle.
// nCyclesIdle should be >= 5.
//RefStat.nSkippedCycles := RefStat.nSkippedCycles + 1;

IF (RefStat.nSkippedCycles >= RefCfg.nMinSkipCycles) THEN
	M_NextMove();
	RefStat.nSkippedCycles:= 0;
END_IF
END_METHOD

METHOD CheckForEvents
VAR_INPUT
END_VAR

VAR
	i:		     INT;
	minState:    INT := 1000;
	maxSubstate: INT := -1000;
END_VAR

nEvent := E_MA_EVENT.HWOK;

IF NOT in_bSafe THEN
	// Not safe to operate the motor
	SetEvent(E_MOTOR_EVENT.UNSAFE);
ELSIF nInternalEvent <> E_MA_EVENT.NONE THEN
	(* Handle internal events *)
	SetEvent(nInternalEvent);
	nInternalEvent := E_MA_EVENT.NONE;
ELSIF RefCtrl.bExecute = TRUE  THEN
	(* Handle commands *)
	RefCtrl.bExecute		:= FALSE;			(* Clear the Execute bit *)
	//M_SetLastCommand(ctrl.nCommand);			(* Save the last command *)
	
	// Device specific log.
	// To be overloaded.
	M_LogCommand();
	
	IF NOT in_bSafe  THEN
		// It is not safe to move motor.
		SetEvent(E_MOTOR_EVENT.UNSAFE);
		M_SetStatus('Unsafe to move motors');
	ELSE
		// WARNING: Here commands are the same as events.
		// Have a look to E_MA_EVENT and E_MA_COMMAND enumerations. They should match!!!
		// This event will be handled by method ProcessEvent
		SetEvent(RefCtrl.nCommand);
	END_IF
	
	RefCtrl.nCommand 		:= E_MA_COMMAND.NONE;	(* Clear the Command *)
ELSIF RefStat.sm.nSubstate = E_MA_SUBSTATE.OP_PRESETTING AND RefStat.bTrackingOK THEN
	// If the system is Presetting and the position error becomes smaller than the threshold,
	// switch to Tracking.
	SetEvent(E_MA_EVENT.PRESETDONE);
	RefCtrl.nCommand 	:= E_MA_COMMAND.NONE;	(* Clear the Command *)
ELSIF RefStat.sm.nSubstate = E_MA_SUBSTATE.OP_TRACKING AND RefStat.bTrackingBAD THEN
	// If the system is Tracking and the position error becomes larger than twice the threshold,
	// switch back to Presetting.
	SetEvent(E_MA_EVENT.TRACKEXIT);
	RefCtrl.nCommand 	:= E_MA_COMMAND.NONE;	(* Clear the Command *)
ELSE
	// Capture unexpected state changes or errors
	FOR i := 1 TO nNumAxes DO
		// Save the minimum state of all axes
		IF (ptrMotorStat[i]^.nState < minState) THEN
			minState := ptrMotorStat[i]^.nState;
		END_IF
		IF (ptrMotorStat[i]^.nSubstate > maxSubstate) THEN
			maxSubstate := ptrMotorStat[i]^.nSubstate;
		END_IF
		// Try to capture a state change when axes are controlled outside the multiaxis.
		// Note: INT_TO_DINT() is used just to be able to compare two variables
		//       of different enumerated type.
		IF	(RefStat.sm.nSubstate <> E_MA_SUBSTATE.OP_DISABLING) AND
			(INT_TO_DINT(ptrMotorStat[i]^.nState) < INT_TO_DINT(RefStat.sm.nState)) THEN
			IF ptrMotorStat[i]^.nState = E_MOTOR_STATE.NOTOP THEN
				SetState(E_MA_STATE.NOTOP, E_MA_SUBSTATE.NOTOP_ERROR);
			ELSE
				SetState(E_MA_STATE.OP, E_MA_SUBSTATE.OP_ERROR);
			END_IF
			M_SetStatus('Unexpected motor state change.');
			RETURN;
		END_IF
		// Capture unexpected motor failure.
		IF (ptrMotorStat[i]^.nSubstate = E_MOTOR_SUBSTATE.OP_ERROR) THEN
			IF RefStat.sm.nState = E_MA_STATE.NOTOP THEN
				SetState(E_MA_STATE.NOTOP, E_MA_SUBSTATE.NOTOP_ERROR);
			ELSE
				SetState(E_MA_STATE.OP, E_MA_SUBSTATE.OP_ERROR);
			END_IF
			M_SetStatus('Unexpected motor error state.');
			RETURN;
		END_IF
    END_FOR
END_IF
END_METHOD

METHOD M_AxesIdle : BOOL
VAR_INPUT
END_VAR
VAR
	i:		INT;
	nState:	INT;
	nSubstate:	INT;
END_VAR
// If any of the motors is not standstill, return FALSE.
FOR i := 1 TO nNumAxes DO
	nState		:= ptrMotorStat[i]^.nState;
	nSubstate	:= ptrMotorStat[i]^.nSubstate;
	
	IF ((nState = E_MOTOR_STATE.NOTOP) AND 
		((nSubstate = E_MA_SUBSTATE.NOTOP_INITIALISING) OR 
		 (nSubstate = E_MA_SUBSTATE.NOTOP_ABORTING))) THEN
		M_AxesIdle	:= FALSE;
		RETURN;
	ELSIF ((nState = E_MOTOR_STATE.OP) AND 
		((nSubstate = E_MA_SUBSTATE.OP_MOVING) OR 
		 (nSubstate = E_MA_SUBSTATE.OP_TRACKING) OR 
		 (nSubstate = E_MA_SUBSTATE.OP_STOPPING))) THEN
		M_AxesIdle	:= FALSE;
		RETURN;
	END_IF
END_FOR

M_AxesIdle	:= TRUE;
END_METHOD

METHOD M_AxesInitialised : BOOL
VAR_INPUT
END_VAR
VAR
	i:		INT;
END_VAR
// If any axis is not initialised, return FALSE.
FOR i := 1 TO nNumAxes DO
	IF NOT ptrMotorStat[i]^.bInitialised THEN
		M_AxesInitialised	:= FALSE;
		RETURN;
	END_IF	
END_FOR

M_AxesInitialised	:= TRUE;
END_METHOD

// Check the state and substate of the motor.
// Returns TRUE if both state and substate match input parameters.
METHOD M_CheckAxesState : BOOL
VAR_INPUT
	in_nState:		E_MOTOR_STATE;
	in_nSubstate:	E_MOTOR_SUBSTATE;
END_VAR
VAR
	i:		INT;
END_VAR
// If any axis state doesn't match, return FALSE.
FOR i := 1 TO nNumAxes DO
	IF (ptrMotorStat[i]^.nState <> in_nState)  OR (ptrMotorStat[i]^.nSubstate <> in_nSubstate) THEN
		M_CheckAxesState	:= FALSE;
		RETURN;
	END_IF	
END_FOR

M_CheckAxesState	:= TRUE;
END_METHOD

METHOD M_CheckError : BOOL
VAR_INPUT
END_VAR
VAR
	i:		INT;
END_VAR
FOR i := 1 TO nNumAxes DO
	IF (ptrMotorStat[i]^.nErrorCode <> E_MOTOR_ERROR.OK) THEN
		M_CheckError	:= TRUE;
		RETURN;
	END_IF	
END_FOR
END_METHOD

METHOD M_Configure : BOOL
VAR_INPUT
END_VAR
VAR
	j:					INT;
	fbGetCurTaskIdx:	GETCURTASKINDEX;
	nCycleTime:			UDINT;END_VAR
VAR_INST
	{attribute 'OPC.UA.DA' := '0'}
	i:	INT := 0;
END_VAR
IF nNumAxes < 1 OR nNumAxes > GPL.C_MA_MAX_AXES THEN
	RefStat.sStatus	:= 'ERROR: Number of axes is not between 2 and 6.';
	RETURN;
END_IF

// Configure the system in stages after boot-up.
// WARNING:
// It seems that setting of pointers takes some time and cannot be done in FB_Init.
// After 40 cycles, we set pointers to motors.
// After 60 cycles, we set pointers to motor sub-structures.
// After 80 cycles, we set general configuration parameters and complete configuration.
IF NOT RefStat.bConfigured THEN
	i	:= i + 1;
	IF i = 40 THEN
		// Assign pointers to the motor device instances
		pMotor[1] := pMotor1;
		pMotor[2] := pMotor2;
		pMotor[3] := pMotor3;
		pMotor[4] := pMotor4;
		pMotor[5] := pMotor5;
		pMotor[6] := pMotor6;
	ELSIF i = 60 THEN
		// Set pointers to motor configuration, control and status.
		// Only set pointers for motors that exist, i.e. != 0.
		FOR j := 1 TO nNumAxes DO
			IF pMotor[j] <> 0 THEN
				ptrMotorCfg[j]	:= ADR(pMotor[j]^.cfg);
				ptrMotorCtrl[j]	:= ADR(pMotor[j]^.ctrl);
				ptrMotorStat[j]	:= ADR(pMotor[j]^.stat);
			ELSE
				RefStat.sStatus	:= 'ERROR: Motor registered but pointer in NULL.';
				i	:= 0;	// Critical error. We must not pass this point.
				RETURN;
			END_IF
		END_FOR
	ELSIF i = 80 THEN

		// Set Motor.library version
		RefStat.sLibVersion	:= Global_Version.stLibVersion_ESO_LDC_Motor_Library.sVersion;
		
		// Get cycle time
		fbGetCurTaskIdx();
		RefStat.nCycleTime := TwinCAT_SystemInfoVarList._TaskInfo[fbGetCurTaskIdx.index].CycleTime;

		// Execute User_Configure().
		User_Configure();
		
		// Create Event instances
		fbEventGeneral.CreateEx	(TC_EVENTS.MotorOpsEventClass.General,0);
		fbEventError.CreateEx	(TC_EVENTS.MotorOpsEventClass.Error,0);

		// We have finished configuration.
		RefStat.bConfigured	:= TRUE;
	END_IF
END_IF
END_METHOD

// Get maximum positioning error of all motors.
// This value should be compared with the 
// threshold for tracking since it takes some time for
// the motors to start following the trajectory properly.
METHOD M_GetMaxPosError : LREAL
VAR_INPUT
END_VAR
VAR
	i: 			INT;
	lrMaxError:	LREAL := 0.0;
	lrError:	LREAL;
END_VAR
FOR i := 1 TO nNumAxes DO
	lrError	:= ABS(ptrMotorStat[i]^.lrPosActual - ptrMotorStat[i]^.lrPosTarget);
	IF lrError > lrMaxError THEN
		lrMaxError := lrError;
	END_IF
END_FOR

M_GetMaxPosError	:= lrMaxError;
END_METHOD

METHOD M_GetRpcErrorText : STRING
VAR_INPUT
	ErrorCode:	INT;
END_VAR
VAR
	str:	STRING;
END_VAR
CASE ErrorCode OF
	E_MOTOR_RPC_ERROR.OK:					str	:= 'OK';
	E_MOTOR_RPC_ERROR.NOT_OP:				str	:= 'Cannot control motor. Not in OP state.';
	E_MOTOR_RPC_ERROR.NOT_NOTOP_READY:		str	:= 'Call failed. Not in NOTOP_READY.';
	E_MOTOR_RPC_ERROR.NOT_NOTOP_NOTREADY:	str	:= 'Call failed. Not in NOTOP_NOTREADY/ERROR.';
	E_MOTOR_RPC_ERROR.LOCAL:				str	:= 'RPC calls not allowed in Local mode.';
	E_MOTOR_RPC_ERROR.SW_LIMIT_LOWER:		str	:= 'Move rejected. Target Pos < Lower SW Limit';
	E_MOTOR_RPC_ERROR.SW_LIMIT_UPPER:		str	:= 'Move rejected. Target Pos > Upper SW Limit';
	E_MOTOR_RPC_ERROR.INIT_WHILE_MOVING:	str	:= 'Cannot INIT moving motor. Motor stopped. Retry.';
	E_MOTOR_RPC_ERROR.VEL_ZERO:				str	:= 'Set velocity cannot be zero';
	E_MOTOR_RPC_ERROR.VEL_NEG:				str	:= 'Set velocity not allowed (<=0)';
	E_MOTOR_RPC_ERROR.VEL_MAX:				str	:= 'Set velocity not allowed (>Vel_max)';
	E_MOTOR_RPC_ERROR.UNSAFE:				str	:= 'Unsafe to move the motor.';
ELSE
	str	:= 'Unregistered RPC error.';
END_CASE

M_GetRpcErrorText	:= str;
END_METHOD

// Move motors. Pos and Vel are already set!
METHOD M_HomeMotors
VAR_INPUT
END_VAR
VAR
	i:			INT;
END_VAR
// Restart timer
M_RestartTimer (RefCfg.timeout.nMoveTimeout);

// Home all axis.
FOR i := 1 TO nNumAxes DO
	ptrMotorCtrl[i]^.lrPosition	:= 0.0;
	ptrMotorCtrl[i]^.lrVelocity	:= ptrMotorCfg[i]^.lrDefaultVelocity;
	ptrMotorCtrl[i]^.nCommand 	:= E_MOTOR_COMMAND.MOTOR_MOVE;
	ptrMotorCtrl[i]^.nMoveType	:= E_MOTOR_MOVE_TYPE.ABSOLUTE;
	ptrMotorCtrl[i]^.bExecute	:= TRUE;
END_FOR
END_METHOD

METHOD M_LogCommand : BOOL
VAR
END_VAR
// Placeholder for MA specific logs, e.g. for DROT or ADC.
// Called in FB_MA_BASE::CheckForEvents():15
END_METHOD

METHOD M_LogEventError : BOOL
VAR_INPUT
	sText:	STRING	:= '';
END_VAR
fbEventError.ipArguments.Clear().AddString(sText);
fbEventError.Send(0);
END_METHOD

METHOD M_LogEventGeneral : BOOL
VAR_INPUT
	sText:	STRING	:= '';
END_VAR
// Log only if logging is enabled AND it is not a tracking command
//IF  NOT cfg.bLog OR ctrl.nMoveType = E_MOTOR_MOVE_TYPE.TRACKING THEN
//	RETURN;
//END_IF

fbEventGeneral.ipArguments.Clear().AddString(sText);
fbEventGeneral.Send(0);
END_METHOD

// Command motors to move to next position.
METHOD M_NextMove
VAR_INPUT
END_VAR
VAR
END_VAR
// Calculate next position for each axes based on the current mode.
User_ComputeNextPos();

// Move axes
ActionTrackExecute();
END_METHOD

// Command motors to move to next position.
METHOD M_NextMoveAbs
VAR_INPUT
END_VAR
VAR
END_VAR
// Calculate next position for each axes based on the current mode.
User_ComputeNextPos();

// Move axes
ActionMoveAbsExecute();
END_METHOD

METHOD M_RestartTimer : BOOL
VAR_INPUT
	in_time:	UDINT := 10000;
END_VAR
// Restart timer
waitTout (IN := FALSE); 				// Reset timer 
waitTout (IN := TRUE, PT := UDINT_TO_TIME(in_time));	// Enable timer
END_METHOD

METHOD M_SetInit
VAR_INPUT
	newState: BOOL;
END_VAR
RefStat.bInitialised := newState;
END_METHOD

METHOD M_SetMode : BOOL
VAR_INPUT
	nMode:	INT;
END_VAR
RefCtrl.nMode	:= nMode;
RefStat.nMode	:= nMode;
END_METHOD

METHOD M_SetRpcStatus : INT
VAR_INPUT
	nErrorCode:	INT;
END_VAR
RefStat.nRpcErrorCode	:= nErrorCode;
RefStat.sRpcErrorText	:= M_GetRpcErrorText(nErrorCode);

M_SetRpcStatus		:= nErrorCode;
END_METHOD

// Set status string
METHOD M_SetStatus : BOOL
VAR_INPUT
	in_sStatus:	STRING	:= '';
END_VAR
RefStat.sStatus	:= in_sStatus;
END_METHOD

METHOD ProcessEvents
VAR_INPUT
END_VAR

RefStat.nSkippedCycles	:= RefStat.nSkippedCycles + 1;

(* 
	Before processing the event, execute the Do-Activity tasks. 
	Note that, in case of orthogonal regions, more than one Do-Activity 
	could run in the same PLC cycle.
	Note: Most of these activities have timeouts since they take time.
*)

IF RefStat.sm.nSubstate = E_MA_SUBSTATE.NOTOP_RESETTING THEN
	ActivityResetting();
END_IF

IF RefStat.sm.nSubstate = E_MA_SUBSTATE.NOTOP_INITIALISING THEN
	ActivityInitialising();
END_IF

IF RefStat.sm.nSubstate = E_MA_SUBSTATE.NOTOP_ENABLING THEN
	ActivityEnabling();
END_IF

IF RefStat.sm.nSubstate = E_MA_SUBSTATE.NOTOP_ABORTING THEN
	ActivityStopping();
END_IF

IF RefStat.sm.nSubstate = E_MA_SUBSTATE.OP_DISABLING THEN
	ActivityDisabling();
END_IF

IF RefStat.sm.nSubstate = E_MA_SUBSTATE.OP_MOVING	AND 
	RefCtrl.nCommand <> E_MA_COMMAND.STOP 				THEN
	ActivityMoving();
END_IF

IF	RefStat.sm.nSubstate = E_MA_SUBSTATE.OP_PRESETTING	AND 
	RefCtrl.nCommand <> E_MA_COMMAND.STOP 				AND 
	RefCtrl.nCommand <> E_MA_COMMAND.STOP_TRACK 			THEN
	ActivityPresetting();
END_IF

IF RefStat.sm.nSubstate = E_MA_SUBSTATE.OP_TRACKING	AND 
	RefCtrl.nCommand <> E_MA_COMMAND.STOP 			AND 
	RefCtrl.nCommand <> E_MA_COMMAND.STOP_TRACK 		 THEN
	ActivityTracking();
END_IF

IF RefStat.sm.nSubstate = E_MA_SUBSTATE.OP_STOPPING THEN
	ActivityStopping();
END_IF

CASE RefStat.sm.nState OF	

  // NotOperational - NotRead case
  E_MA_STATE.NOTOP:	
	  CASE nEvent OF
		  E_MA_EVENT.RESET:
			  ActionResetExecute();
			  SetState(E_MA_STATE.NOTOP, E_MA_SUBSTATE.NOTOP_RESETTING);
		  E_MA_EVENT.INIT:
			  ActionInitExecute();
			  SetState(E_MA_STATE.NOTOP, E_MA_SUBSTATE.NOTOP_INITIALISING);
		  E_MA_EVENT.ENABLE: 
			  ActionEnableExecute();
			  SetState(E_MA_STATE.NOTOP, E_MA_SUBSTATE.NOTOP_ENABLING);
		  E_MA_EVENT.STOP:
			  ActionStopExecute();
			  SetState(E_MA_STATE.NOTOP, E_MA_SUBSTATE.NOTOP_ABORTING);
	      E_MA_EVENT.STOP_TRACK:
		        M_SetStatus('ERROR: controller is not Operational');
			E_MA_EVENT.MA_MOVE:
				M_SetStatus('ERROR: controller is not Operational');
			E_MA_EVENT.START_TRACK:
				M_SetStatus('ERROR: controller is not Operational');
	  END_CASE
		
  // Operational case //
  E_MA_STATE.OP:
       CASE nEvent OF
			E_MA_EVENT.DISABLE: 
				THIS^.ActionDisableExecute();
				SetState(E_MA_STATE.OP, E_MA_SUBSTATE.OP_DISABLING);
				
			E_MA_EVENT.RESET: 
				THIS^.ActionResetExecute();
				SetState(E_MA_STATE.NOTOP, E_MA_SUBSTATE.NOTOP_RESETTING);
				
			E_MA_EVENT.STOP:
				// Stop the motor at current position, whatever it is.
				RefStat.nSkippedCycles 	:= RefCfg.nMinSkipCycles + 1; // Immediate action
				M_SetMode(E_MA_MODE.MA_MODE_ENG);
				ActionStopExecute();
				SetState(E_MA_STATE.OP, E_MA_SUBSTATE.OP_STOPPING);
				
			E_MA_EVENT.STOP_TRACK:
				M_SetMode(RefCtrl.nMode);	
				// Set nCyclesIdle to zero.
				// Needed to distinguish if the motor is about to move off or it completed the move.
//				RefStat.nSkippedCycles 	:= 0;	// Delayed action
				RefStat.nSkippedCycles 	:= RefCfg.nMinSkipCycles + 1; // Immediate action
				M_NextMoveAbs();
				SetState(E_MA_STATE.OP, E_MA_SUBSTATE.OP_MOVING);
				
